ABB RobotStudio station: powerpac.rsstn

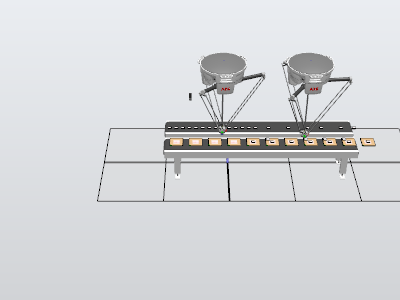
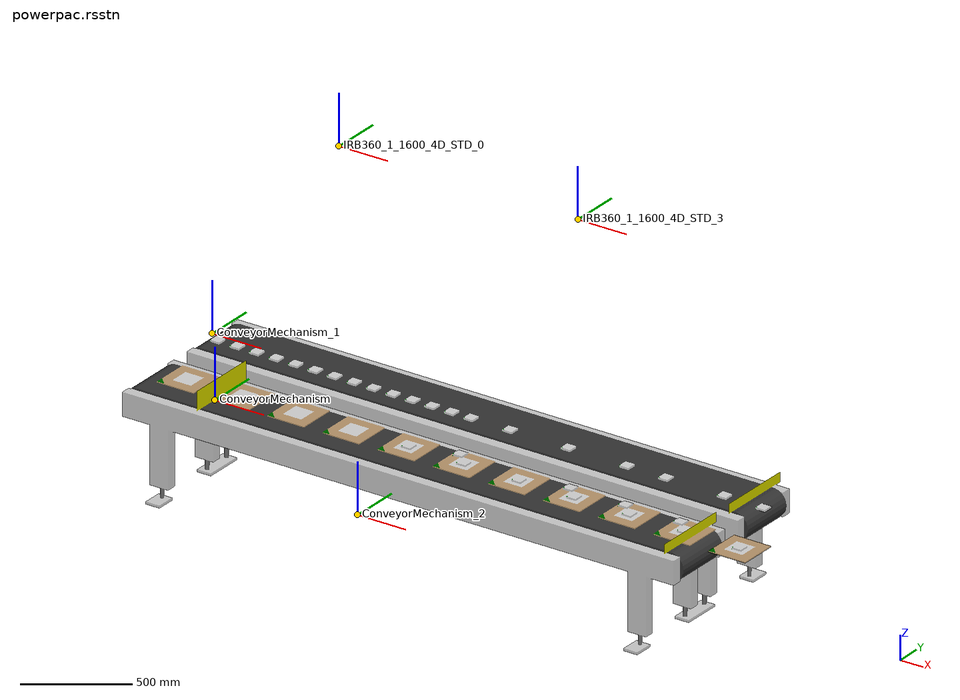
[picture v1: parts stored in the station drawn from their meshes, with robot base, taught points and paths (robot models come from the ABB library and are not in the file)]
Station Station (saved by RobotStudio 22.3.10141.1)
Controller Controller5, task T_ROB1: task frame (RAPID world) sits at (1200, 0, 1800) mm in the station
Controller Controller4, task T_ROB1: task frame (RAPID world) sits at (-100, 0, 1800) mm in the station
Controller Controller4
  mechanical unit ROB_1: IRB360_1_1600_4D_STD_02, 4 joints, base frame (0, 0, 0) mm, rotated rx 180 ry 0 rz 0 deg
  mechanical unit CNV2: ConveyorMechanism, 1 joints, base frame (-500, -250, -1300) mm
  mechanical unit CNV1: ConveyorMechanism_1, 1 joints, base frame (-900, 300, -1300) mm
Controller Controller5
  mechanical unit ROB_1: IRB360_1_1600_4D_STD_3, 4 joints, base frame (0, 0, 0) mm, rotated rx 180 ry 0 rz 0 deg
  mechanical unit CNV2: ConveyorMechanism_2, 1 joints, base frame (0, 0, 0) mm
  mechanical unit CNV1: ConveyorMechanism_3, 1 joints, base frame (0, 0, 0) mm
Layout (positions relative to the parent item):
  - IRB360_1_1600_4D_STD_02 [mechanism, from Robots\IRB360_1_1600_4D_STD_02.rslib] at (-100, 0, 1800) mm, rotated rx 180 ry 0 rz 0 deg; joint values [-0.192, -0.192, -0.192, 0] (rad or m)
  - Line [smart component]
      properties: Enabled=true
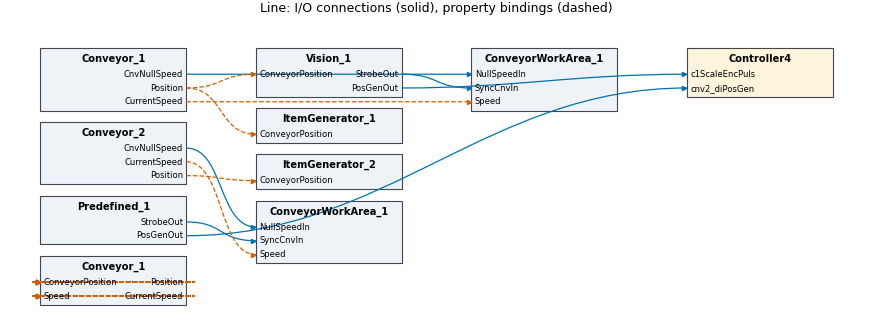
      connections:
        Conveyor_1.CnvNullSpeed -> ConveyorWorkArea_1.NullSpeedIn
        Conveyor_2.CnvNullSpeed -> ConveyorWorkArea_1.NullSpeedIn
        Vision_1.StrobeOut -> ConveyorWorkArea_1.SyncCnvIn
        Vision_1.PosGenOut -> Controller4.c1ScaleEncPuls
        Predefined_1.StrobeOut -> ConveyorWorkArea_1.SyncCnvIn
        Predefined_1.PosGenOut -> Controller4.cnv2_diPosGen
        Conveyor_1.Position => Vision_1.ConveyorPosition
        Conveyor_1.CurrentSpeed => ConveyorWorkArea_1.Speed
        Conveyor_1.Position => ItemGenerator_1.ConveyorPosition
        Conveyor_2.Position => ItemGenerator_2.ConveyorPosition
        Conveyor_1.Position => Vision_1.ConveyorPosition
        Conveyor_1.CurrentSpeed => ConveyorWorkArea_1.Speed
        Conveyor_1.Position => ItemGenerator_1.ConveyorPosition
        Conveyor_2.Position => ItemGenerator_2.ConveyorPosition
        Conveyor_1.Position => Vision_1.ConveyorPosition
        Conveyor_1.CurrentSpeed => ConveyorWorkArea_1.Speed
        Conveyor_2.CurrentSpeed => ConveyorWorkArea_1.Speed
        Conveyor_1.Position => ItemGenerator_1.ConveyorPosition
        Conveyor_2.Position => ItemGenerator_2.ConveyorPosition
        Conveyor_1.Position => Vision_1.ConveyorPosition
        Conveyor_1.CurrentSpeed => ConveyorWorkArea_1.Speed
        Conveyor_2.CurrentSpeed => ConveyorWorkArea_1.Speed
        Conveyor_1.Position => ItemGenerator_1.ConveyorPosition
        Conveyor_2.Position => ItemGenerator_2.ConveyorPosition
        Conveyor_1.Position => Vision_1.ConveyorPosition
        Conveyor_1.CurrentSpeed => ConveyorWorkArea_1.Speed
        Conveyor_2.CurrentSpeed => ConveyorWorkArea_1.Speed
        Conveyor_1.Position => ItemGenerator_1.ConveyorPosition
        Conveyor_2.Position => ItemGenerator_2.ConveyorPosition
        Conveyor_1.Position => Vision_1.ConveyorPosition
        Conveyor_1.CurrentSpeed => ConveyorWorkArea_1.Speed
        Conveyor_2.CurrentSpeed => ConveyorWorkArea_1.Speed
        Conveyor_1.Position => ItemGenerator_1.ConveyorPosition
        Conveyor_2.Position => ItemGenerator_2.ConveyorPosition
    - Job_1 [smart component]
        properties: Project=C:\Users\aedpu\OneDrive\Documents\RobotStudio\Picking\PMPPProject.pmproj; Enabled=true; UserName=admin; Password=password
      - ItemGenerator_1 [smart component]
          properties: ItemSource=Item_1; PositionSource=Vision_1; Conveyor=Conveyor_1; Offset=[[1 0 0 0] [0 1 0 0] [0 0 1 0] [-1 0.250000005960464 0.5 1]]; ObjectLocation=[0.00273041710121014 0 0]; ObjectOrientation=[0 0 0]; ItemContainer=MotionContainer; ConveyorPosition=8.22780232501204; TriggerDistance=0.105999998748302; ProductInfos=1 True 0 0 0 0 0 0;; Repeat=true; Stability=100; OrientationStability=100; ZOriDevMin=0; ZOriDevMax=0; RejectionRatio=0; PositionStability=100; XPosDevMin=0; XPosDevMax=0; YPosDevMin=0; YPosDevMax=0
          signals: DO ItemCreated, DI ItemCopied, DI QueueIdleIn, DI GenerateItemsIn, DO GenerateItemsOut, DI GenerateMultipleItemsIn
          connections:
            ItemGenerator_1.GenerateItemsIn -> ItemGenerator_1.GenerateItemsOut
            ItemGenerator_1.GenerateItemsOut -> ItemCopier.Execute
            ItemCopier.Executed -> ItemGenerator_1.ItemCopied
            ItemCopier.Executed -> ItemCounter.Increase
            CountComparer.Output -> ItemGenerator_1.ItemCreated
            ItemGenerator_1.QueueIdleIn -> Inverter.Input
            Inverter.OutputLow -> ItemCounter.Reset
            ItemGenerator_1.ItemSource => ItemCopier.Source
            ItemGenerator_1.ItemContainer => ItemCopier.Parent
            ItemCounter.Count => CountComparer.ValueA
        - ItemCopier [smart component, from Components\Source.rslib]
            properties: Source=Item_1; Copy=Item_1_1803; Parent=MotionContainer; Position=[0 0 0]; Orientation=[0 0 0]; Transient=false; PhysicsBehavior=0
        - ItemCounter [smart component, from Components\Counter.rslib]
            properties: Count=77
        - CountComparer [smart component, from Components\Comparer.rslib]
            properties: ValueA=77; Operator=>; ValueB=0
        - Inverter [smart component, from Components\LogicSplit.rslib]
      - ItemGenerator_2 [smart component]
          properties: ItemSource=Container_1; PositionSource=Predefined_1; Conveyor=Conveyor_2; Offset=[[1 0 0 0] [0 1 0 0] [0 0 1 0] [-1 -0.249999994039536 0.5 1]]; ObjectLocation=[0.00292999639970226 0 0]; ObjectOrientation=[0 0 0]; ItemContainer=MotionContainer; ConveyorPosition=8.18460232329542; TriggerDistance=0.300000011920929; ProductInfos=1 True 0 0 0 0 0 0;; Repeat=true; Stability=100; OrientationStability=100; ZOriDevMin=0; ZOriDevMax=0; RejectionRatio=0; PositionStability=100; XPosDevMin=0; XPosDevMax=0; YPosDevMin=0; YPosDevMax=0
          signals: DO ItemCreated, DI ItemCopied, DI QueueIdleIn, DI GenerateItemsIn, DO GenerateItemsOut, DI GenerateMultipleItemsIn
          connections:
            ItemGenerator_2.GenerateItemsIn -> ItemGenerator_2.GenerateItemsOut
            ItemGenerator_2.GenerateItemsOut -> ItemCopier.Execute
            ItemCopier.Executed -> ItemGenerator_2.ItemCopied
            ItemCopier.Executed -> ItemCounter.Increase
            CountComparer.Output -> ItemGenerator_2.ItemCreated
            ItemGenerator_2.QueueIdleIn -> Inverter.Input
            Inverter.OutputLow -> ItemCounter.Reset
            ItemGenerator_2.ItemSource => ItemCopier.Source
            ItemGenerator_2.ItemContainer => ItemCopier.Parent
            ItemCounter.Count => CountComparer.ValueA
        - ItemCopier [smart component, from Components\Source.rslib]
            properties: Source=Container_1; Copy=Container_1_1804; Parent=MotionContainer; Position=[0 0 0]; Orientation=[0 0 0]; Transient=false; PhysicsBehavior=0
        - ItemCounter [smart component, from Components\Counter.rslib]
            properties: Count=27
        - CountComparer [smart component, from Components\Comparer.rslib]
            properties: ValueA=27; Operator=>; ValueB=0
        - Inverter [smart component, from Components\LogicSplit.rslib]
    - PickPlaceTool_1 [smart component, from %3FC1A3B3-DC1B-42D2-8AA6-D9E1B3C46536%\PMPickPlaceTool.rslib] at (-100, 0, 623.14) mm, rotated rx 180 ry 0 rz 0 deg
        properties: AttachLocation=[0 0 0.07]; AttachOrientation=[3.14159265358979 0 0]; PickLimit=0.05; PlaceLimit=0.1; GripSignal=doVacuum1; ReleaseSignal=doBlow1
        connections:
          PickPlaceTool_1.GripIn -> PickPlaceTool_1.GripOut
          PickPlaceTool_1.ReleaseIn -> PickPlaceTool_1.ReleaseOut
    - PickPlaceTool_2 [smart component, from %3FC1A3B3-DC1B-42D2-8AA6-D9E1B3C46536%\PMPickPlaceTool.rslib] at (1200, 0, 545.63) mm, rotated rx 180 ry 0 rz 0 deg
        properties: AttachLocation=[0 0 0.07]; AttachOrientation=[3.14159265358979 0 0]; PickLimit=0.05; PlaceLimit=0.1; GripSignal=doVacuum1; ReleaseSignal=doBlow1
        connections:
          PickPlaceTool_2.GripIn -> PickPlaceTool_2.GripOut
          PickPlaceTool_2.ReleaseIn -> PickPlaceTool_2.ReleaseOut
    - Vision_1 [smart component, from %3FC1A3B3-DC1B-42D2-8AA6-D9E1B3C46536%\PMVision.rslib] at (-600, 300, 1000) mm
        properties: Id=213262b1-3477-4070-b768-c16ae12cfddf; Entry=-0.2; Exit=0.2; Left=-0.2; Right=0.2; LimitVisionWidth=false; TriggerType=Distance; TriggerDistance=0.150000005960464; PositionDelay=0; ConveyorPosition=8.22780232501204; SpotLight=Camera 1; PlaneSensor=(none)
        connections:
          Vision_1.TrigVisionIn -> Vision_1.StrobeOut
          Vision_1.PosGenIn -> Vision_1.PosGenOut
    - Conveyor_1 [smart component] at (-1000, 300, 500) mm
        properties: CalibrationLocation=[0 0 0]; CalibrationOrientation=[0 0 0]; Length=3; Width=0.400000005960464; Exit=3; Speed=0.300000011920929; Acc=0.5; Dec=1; CurrentSpeed=0; Position=8.22780232501204; SpeedSignal=; IOMapSystemId=
        signals: DI CnvStartStopIn, DO CnvStartStopOut, DO CnvNullSpeed, AI CnvSpeed
        connections:
          Conveyor_1.CnvStartStopIn -> Conveyor_1.CnvStartStopOut
          ConveyorWorkArea_1.Cnt1FromEncOut -> Controller4.CNV1_giCntSim
          ConveyorWorkArea_1.ConnectedOut -> Controller4.c1Connected
          ConveyorWorkArea_1.NewObjStrobeOut -> Controller4.c1NewObjStrobe
          ConveyorWorkArea_1.PositionOut -> Controller4.c1Position
          ConveyorWorkArea_1.SpeedOut -> Controller4.c1Speed
          ConveyorWorkArea_1.NullSpeedOut -> Controller4.c1NullSpeed
          Conveyor_1.CurrentSpeed => Mover.Speed
          Conveyor_1.Exit => ExitHandler.Transform.X
      - MotionContainer [graphiccomponentgroup] at (8227.8, 0, 0) mm
        - Item_1_1766 [smart component] at (-5194, -50, 0) mm
            properties: Id=2704d276-ea2d-4d5a-9f22-027de52e7f75; GripLocation=[0 0 0.01]; GripOrientation=[0 0 0]; Assembled=true; Detect=true; Accepted=true; IgnoreOrientation=false
          - Item1 [graphiccomponentgroup]
            - MainBody [part], size 50 x 50 x 10 mm
            - OuterLine [part], size 50 x 50 x 10 mm
            - Labels [part], size 25 x 25 x 0 mm
            - Origin [part], size 10.5 x 10.5 x 11 mm
            - RejectSymbol [part], size 23.8 x 48.1 x 1 mm
        - Item_1_1768 [smart component] at (-5406, -50, 0) mm
            properties: Id=2704d276-ea2d-4d5a-9f22-027de52e7f75; GripLocation=[0 0 0.01]; GripOrientation=[0 0 0]; Assembled=true; Detect=true; Accepted=true; IgnoreOrientation=false
          - Item1 [graphiccomponentgroup]
            - MainBody [part], size 50 x 50 x 10 mm
            - OuterLine [part], size 50 x 50 x 10 mm
            - Labels [part], size 25 x 25 x 0 mm
            - Origin [part], size 10.5 x 10.5 x 11 mm
            - RejectSymbol [part], size 23.8 x 48.1 x 1 mm
        - Item_1_1772 [smart component] at (-5724, -50, 0) mm
            properties: Id=2704d276-ea2d-4d5a-9f22-027de52e7f75; GripLocation=[0 0 0.01]; GripOrientation=[0 0 0]; Assembled=true; Detect=true; Accepted=true; IgnoreOrientation=false
          - Item1 [graphiccomponentgroup]
            - MainBody [part], size 50 x 50 x 10 mm
            - OuterLine [part], size 50 x 50 x 10 mm
            - Labels [part], size 25 x 25 x 0 mm
            - Origin [part], size 10.5 x 10.5 x 11 mm
            - RejectSymbol [part], size 23.8 x 48.1 x 1 mm
        - Item_1_1775 [smart component] at (-5936, -50, 0) mm
            properties: Id=2704d276-ea2d-4d5a-9f22-027de52e7f75; GripLocation=[0 0 0.01]; GripOrientation=[0 0 0]; Assembled=true; Detect=true; Accepted=true; IgnoreOrientation=false
          - Item1 [graphiccomponentgroup]
            - MainBody [part], size 50 x 50 x 10 mm
            - OuterLine [part], size 50 x 50 x 10 mm
            - Labels [part], size 25 x 25 x 0 mm
            - Origin [part], size 10.5 x 10.5 x 11 mm
            - RejectSymbol [part], size 23.8 x 48.1 x 1 mm
        - Item_1_1779 [smart component] at (-6254, -50, 0) mm
            properties: Id=2704d276-ea2d-4d5a-9f22-027de52e7f75; GripLocation=[0 0 0.01]; GripOrientation=[0 0 0]; Assembled=true; Detect=true; Accepted=true; IgnoreOrientation=false
          - Item1 [graphiccomponentgroup]
            - MainBody [part], size 50 x 50 x 10 mm
            - OuterLine [part], size 50 x 50 x 10 mm
            - Labels [part], size 25 x 25 x 0 mm
            - Origin [part], size 10.5 x 10.5 x 11 mm
            - RejectSymbol [part], size 23.8 x 48.1 x 1 mm
        - Item_1_1783 [smart component] at (-6572, -50, 0) mm
            properties: Id=2704d276-ea2d-4d5a-9f22-027de52e7f75; GripLocation=[0 0 0.01]; GripOrientation=[0 0 0]; Assembled=true; Detect=true; Accepted=true; IgnoreOrientation=false
          - Item1 [graphiccomponentgroup]
            - MainBody [part], size 50 x 50 x 10 mm
            - OuterLine [part], size 50 x 50 x 10 mm
            - Labels [part], size 25 x 25 x 0 mm
            - Origin [part], size 10.5 x 10.5 x 11 mm
            - RejectSymbol [part], size 23.8 x 48.1 x 1 mm
        - Item_1_1786 [smart component] at (-6784, -50, 0) mm
            properties: Id=2704d276-ea2d-4d5a-9f22-027de52e7f75; GripLocation=[0 0 0.01]; GripOrientation=[0 0 0]; Assembled=true; Detect=true; Accepted=true; IgnoreOrientation=false
          - Item1 [graphiccomponentgroup]
            - MainBody [part], size 50 x 50 x 10 mm
            - OuterLine [part], size 50 x 50 x 10 mm
            - Labels [part], size 25 x 25 x 0 mm
            - Origin [part], size 10.5 x 10.5 x 11 mm
            - RejectSymbol [part], size 23.8 x 48.1 x 1 mm
        - Item_1_1787 [smart component] at (-6890, -50, 0) mm
            properties: Id=2704d276-ea2d-4d5a-9f22-027de52e7f75; GripLocation=[0 0 0.01]; GripOrientation=[0 0 0]; Assembled=true; Detect=true; Accepted=true; IgnoreOrientation=false
          - Item1 [graphiccomponentgroup]
            - MainBody [part], size 50 x 50 x 10 mm
            - OuterLine [part], size 50 x 50 x 10 mm
            - Labels [part], size 25 x 25 x 0 mm
            - Origin [part], size 10.5 x 10.5 x 11 mm
            - RejectSymbol [part], size 23.8 x 48.1 x 1 mm
        - Item_1_1789 [smart component] at (-6996, -50, 0) mm
            properties: Id=2704d276-ea2d-4d5a-9f22-027de52e7f75; GripLocation=[0 0 0.01]; GripOrientation=[0 0 0]; Assembled=true; Detect=true; Accepted=true; IgnoreOrientation=false
          - Item1 [graphiccomponentgroup]
            - MainBody [part], size 50 x 50 x 10 mm
            - OuterLine [part], size 50 x 50 x 10 mm
            - Labels [part], size 25 x 25 x 0 mm
            - Origin [part], size 10.5 x 10.5 x 11 mm
            - RejectSymbol [part], size 23.8 x 48.1 x 1 mm
        - Item_1_1790 [smart component] at (-7102, -50, 0) mm
            properties: Id=2704d276-ea2d-4d5a-9f22-027de52e7f75; GripLocation=[0 0 0.01]; GripOrientation=[0 0 0]; Assembled=true; Detect=true; Accepted=true; IgnoreOrientation=false
          - Item1 [graphiccomponentgroup]
            - MainBody [part], size 50 x 50 x 10 mm
            - OuterLine [part], size 50 x 50 x 10 mm
            - Labels [part], size 25 x 25 x 0 mm
            - Origin [part], size 10.5 x 10.5 x 11 mm
            - RejectSymbol [part], size 23.8 x 48.1 x 1 mm
        - Item_1_1791 [smart component] at (-7208, -50, 0) mm
            properties: Id=2704d276-ea2d-4d5a-9f22-027de52e7f75; GripLocation=[0 0 0.01]; GripOrientation=[0 0 0]; Assembled=true; Detect=true; Accepted=true; IgnoreOrientation=false
          - Item1 [graphiccomponentgroup]
            - MainBody [part], size 50 x 50 x 10 mm
            - OuterLine [part], size 50 x 50 x 10 mm
            - Labels [part], size 25 x 25 x 0 mm
            - Origin [part], size 10.5 x 10.5 x 11 mm
            - RejectSymbol [part], size 23.8 x 48.1 x 1 mm
        - Item_1_1793 [smart component] at (-7314, -50, 0) mm
            properties: Id=2704d276-ea2d-4d5a-9f22-027de52e7f75; GripLocation=[0 0 0.01]; GripOrientation=[0 0 0]; Assembled=true; Detect=true; Accepted=true; IgnoreOrientation=false
          - Item1 [graphiccomponentgroup]
            - MainBody [part], size 50 x 50 x 10 mm
            - OuterLine [part], size 50 x 50 x 10 mm
            - Labels [part], size 25 x 25 x 0 mm
            - Origin [part], size 10.5 x 10.5 x 11 mm
            - RejectSymbol [part], size 23.8 x 48.1 x 1 mm
        - Item_1_1794 [smart component] at (-7420, -50, 0) mm
            properties: Id=2704d276-ea2d-4d5a-9f22-027de52e7f75; GripLocation=[0 0 0.01]; GripOrientation=[0 0 0]; Assembled=true; Detect=true; Accepted=true; IgnoreOrientation=false
          - Item1 [graphiccomponentgroup]
            - MainBody [part], size 50 x 50 x 10 mm
            - OuterLine [part], size 50 x 50 x 10 mm
            - Labels [part], size 25 x 25 x 0 mm
            - Origin [part], size 10.5 x 10.5 x 11 mm
            - RejectSymbol [part], size 23.8 x 48.1 x 1 mm
        - Item_1_1795 [smart component] at (-7526, -50, 0) mm
            properties: Id=2704d276-ea2d-4d5a-9f22-027de52e7f75; GripLocation=[0 0 0.01]; GripOrientation=[0 0 0]; Assembled=true; Detect=true; Accepted=true; IgnoreOrientation=false
          - Item1 [graphiccomponentgroup]
            - MainBody [part], size 50 x 50 x 10 mm
            - OuterLine [part], size 50 x 50 x 10 mm
            - Labels [part], size 25 x 25 x 0 mm
            - Origin [part], size 10.5 x 10.5 x 11 mm
            - RejectSymbol [part], size 23.8 x 48.1 x 1 mm
        - Item_1_1797 [smart component] at (-7632, -50, 0) mm
            properties: Id=2704d276-ea2d-4d5a-9f22-027de52e7f75; GripLocation=[0 0 0.01]; GripOrientation=[0 0 0]; Assembled=true; Detect=true; Accepted=true; IgnoreOrientation=false
          - Item1 [graphiccomponentgroup]
            - MainBody [part], size 50 x 50 x 10 mm
            - OuterLine [part], size 50 x 50 x 10 mm
            - Labels [part], size 25 x 25 x 0 mm
            - Origin [part], size 10.5 x 10.5 x 11 mm
            - RejectSymbol [part], size 23.8 x 48.1 x 1 mm
        - Item_1_1798 [smart component] at (-7738, -50, 0) mm
            properties: Id=2704d276-ea2d-4d5a-9f22-027de52e7f75; GripLocation=[0 0 0.01]; GripOrientation=[0 0 0]; Assembled=true; Detect=true; Accepted=true; IgnoreOrientation=false
          - Item1 [graphiccomponentgroup]
            - MainBody [part], size 50 x 50 x 10 mm
            - OuterLine [part], size 50 x 50 x 10 mm
            - Labels [part], size 25 x 25 x 0 mm
            - Origin [part], size 10.5 x 10.5 x 11 mm
            - RejectSymbol [part], size 23.8 x 48.1 x 1 mm
        - Item_1_1799 [smart component] at (-7844, -50, 0) mm
            properties: Id=2704d276-ea2d-4d5a-9f22-027de52e7f75; GripLocation=[0 0 0.01]; GripOrientation=[0 0 0]; Assembled=true; Detect=true; Accepted=true; IgnoreOrientation=false
          - Item1 [graphiccomponentgroup]
            - MainBody [part], size 50 x 50 x 10 mm
            - OuterLine [part], size 50 x 50 x 10 mm
            - Labels [part], size 25 x 25 x 0 mm
            - Origin [part], size 10.5 x 10.5 x 11 mm
            - RejectSymbol [part], size 23.8 x 48.1 x 1 mm
        - Item_1_1801 [smart component] at (-7950, -50, 0) mm
            properties: Id=2704d276-ea2d-4d5a-9f22-027de52e7f75; GripLocation=[0 0 0.01]; GripOrientation=[0 0 0]; Assembled=true; Detect=true; Accepted=true; IgnoreOrientation=false
          - Item1 [graphiccomponentgroup]
            - MainBody [part], size 50 x 50 x 10 mm
            - OuterLine [part], size 50 x 50 x 10 mm
            - Labels [part], size 25 x 25 x 0 mm
            - Origin [part], size 10.5 x 10.5 x 11 mm
            - RejectSymbol [part], size 23.8 x 48.1 x 1 mm
        - Item_1_1802 [smart component] at (-8056, -50, 0) mm
            properties: Id=2704d276-ea2d-4d5a-9f22-027de52e7f75; GripLocation=[0 0 0.01]; GripOrientation=[0 0 0]; Assembled=true; Detect=true; Accepted=true; IgnoreOrientation=false
          - Item1 [graphiccomponentgroup]
            - MainBody [part], size 50 x 50 x 10 mm
            - OuterLine [part], size 50 x 50 x 10 mm
            - Labels [part], size 25 x 25 x 0 mm
            - Origin [part], size 10.5 x 10.5 x 11 mm
            - RejectSymbol [part], size 23.8 x 48.1 x 1 mm
        - Item_1_1803 [smart component] at (-8162, -50, 0) mm
            properties: Id=2704d276-ea2d-4d5a-9f22-027de52e7f75; GripLocation=[0 0 0.01]; GripOrientation=[0 0 0]; Assembled=true; Detect=true; Accepted=true; IgnoreOrientation=false
          - Item1 [graphiccomponentgroup]
            - MainBody [part], size 50 x 50 x 10 mm
            - OuterLine [part], size 50 x 50 x 10 mm
            - Labels [part], size 25 x 25 x 0 mm
            - Origin [part], size 10.5 x 10.5 x 11 mm
            - RejectSymbol [part], size 23.8 x 48.1 x 1 mm
      - Mover [smart component, from Components\LinearMover.rslib]
          properties: Object=MotionContainer; Direction=[0.001 0 0]; Speed=0; Reference=Local; ReferenceObject=(none)
      - ExitHandler [smart component, from %3FC1A3B3-DC1B-42D2-8AA6-D9E1B3C46536%\PMExitHandler.rslib] at (3000, 0, 0) mm
          properties: Count=32; SensedObject=(none)
          connections:
            Timer.Output -> ExitHandler.Execute
        - Timer [smart component, from Components\Timer.rslib]
            properties: StartTime=0; Interval=1; Repeat=true; CurrentTime=32.64
      - ConveyorWorkArea_1 [smart component, from %3FC1A3B3-DC1B-42D2-8AA6-D9E1B3C46536%\PMConveyorWorkArea.rslib]
          properties: WorkAreaType=Pick; PositionSource=Vision_1; PositionGeneratorSignal=cnv1_diPosGen; TrigVisionSignal=cnv1_doTrigVis; CnvStartStopSignal=cnv1_doStartCnv; ControllerMechUnit=CNV1; SystemId={3445A632-8DB2-4EAE-9C35-B4E87A875A90}; Speed=0; QueueIdleSignal=cnv1_doQIdle; CountsPerMeter=20000
          connections:
            Converter.AnalogOutput -> ConveyorWorkArea_1.SpeedIn
            ConveyorWorkArea_1.SpeedIn -> ConveyorWorkArea_1.SpeedOut
            ConveyorWorkArea_1.NullSpeedIn -> ConveyorWorkArea_1.NullSpeedOut
            ConveyorWorkArea_1.Speed => Converter.AnalogProperty
        - Converter [smart component, from Components\Converter.rslib]
            properties: AnalogProperty=0; DigitalProperty=0; BooleanProperty=false; GroupProperty=0
    - Predefined_1 [smart component, from %3FC1A3B3-DC1B-42D2-8AA6-D9E1B3C46536%\PMPredefined.rslib]
        properties: Id=fbd0e5b6-92fc-4816-a2a1-f9a7d29e2a65; TriggerType=IO; TriggerDistance=0; ConveyorPosition=0; PlaneSensor=PlaneSensor
        connections:
          Predefined_1.PosGenIn -> Predefined_1.PosGenOut
          Predefined_1.PosGenIn -> Predefined_1.StrobeOut
    - Conveyor_2 [smart component] at (-1000, -200, 500) mm
        properties: CalibrationLocation=[0 0 0]; CalibrationOrientation=[0 0 0]; Length=3; Width=0.400000005960464; Exit=3; Speed=0.300000011920929; Acc=0.5; Dec=1; CurrentSpeed=0; Position=8.18460232329542; SpeedSignal=; IOMapSystemId=
        signals: DI CnvStartStopIn, DO CnvStartStopOut, DO CnvNullSpeed, AI CnvSpeed
        connections:
          Conveyor_2.CnvStartStopIn -> Conveyor_2.CnvStartStopOut
          ConveyorWorkArea_1.Cnt1FromEncOut -> Controller4.CNV2_giCntSim
          ConveyorWorkArea_1.ConnectedOut -> Controller4.c2Connected
          ConveyorWorkArea_1.NewObjStrobeOut -> Controller4.c2NewObjStrobe
          ConveyorWorkArea_1.PositionOut -> Controller4.c2Position
          ConveyorWorkArea_1.SpeedOut -> Controller4.c2Speed
          ConveyorWorkArea_1.NullSpeedOut -> Controller4.c2NullSpeed
          Conveyor_2.CurrentSpeed => Mover.Speed
          Conveyor_2.Exit => ExitHandler.Transform.X
      - MotionContainer [graphiccomponentgroup] at (8184.6, 0, 0) mm
        - Container_1_1765 [smart component] at (-5100, -50, 0) mm
            properties: Id=73001933-2678-449b-9029-7b770ab6b154; GripLocation=[0.1 0.1 0.1]; GripOrientation=[0 0 0]; Detect=true; Accepted=true; IgnoreOrientation=false
          - Container1 [graphiccomponentgroup]
            - MainBody [part], size 200 x 200 x 5 mm
            - OuterLine [part], size 200 x 200 x 5 mm
            - Labels [part], size 100 x 100 x 0 mm
            - Origin [part], size 40.5 x 40.5 x 6 mm
            - RejectSymbol [part], size 47.5 x 96.2 x 1 mm
          - Layer_1 [smart component, from %3FC1A3B3-DC1B-42D2-8AA6-D9E1B3C46536%\PMLayer.rslib] at (0, 0, 5) mm
              properties: Pattern=Pattern_1
          - Layer_2 [smart component, from %3FC1A3B3-DC1B-42D2-8AA6-D9E1B3C46536%\PMLayer.rslib] at (0, 0, 15) mm
              properties: Pattern=Pattern_2
          - Item_1_1763 [smart component] at (101.26, 97.68, 5) mm
              properties: Id=2704d276-ea2d-4d5a-9f22-027de52e7f75; GripLocation=[0 0 0.01]; GripOrientation=[0 0 0]; Assembled=true; Detect=true; Accepted=true; IgnoreOrientation=false
            - Item1 [graphiccomponentgroup]
              - MainBody [part], size 50 x 50 x 10 mm
              - OuterLine [part], size 50 x 50 x 10 mm
              - Labels [part], size 25 x 25 x 0 mm
              - Origin [part], size 10.5 x 10.5 x 11 mm
              - RejectSymbol [part], size 23.8 x 48.1 x 1 mm
        - Container_1_1769 [smart component] at (-5400, -50, 0) mm
            properties: Id=73001933-2678-449b-9029-7b770ab6b154; GripLocation=[0.1 0.1 0.1]; GripOrientation=[0 0 0]; Detect=true; Accepted=true; IgnoreOrientation=false
          - Container1 [graphiccomponentgroup]
            - MainBody [part], size 200 x 200 x 5 mm
            - OuterLine [part], size 200 x 200 x 5 mm
            - Labels [part], size 100 x 100 x 0 mm
            - Origin [part], size 40.5 x 40.5 x 6 mm
            - RejectSymbol [part], size 47.5 x 96.2 x 1 mm
          - Layer_1 [smart component, from %3FC1A3B3-DC1B-42D2-8AA6-D9E1B3C46536%\PMLayer.rslib] at (0, 0, 5) mm
              properties: Pattern=Pattern_1
          - Layer_2 [smart component, from %3FC1A3B3-DC1B-42D2-8AA6-D9E1B3C46536%\PMLayer.rslib] at (0, 0, 15) mm
              properties: Pattern=Pattern_2
          - Item_1_1764 [smart component] at (101.26, 97.68, 5) mm
              properties: Id=2704d276-ea2d-4d5a-9f22-027de52e7f75; GripLocation=[0 0 0.01]; GripOrientation=[0 0 0]; Assembled=true; Detect=true; Accepted=true; IgnoreOrientation=false
            - Item1 [graphiccomponentgroup]
              - MainBody [part], size 50 x 50 x 10 mm
              - OuterLine [part], size 50 x 50 x 10 mm
              - Labels [part], size 25 x 25 x 0 mm
              - Origin [part], size 10.5 x 10.5 x 11 mm
              - RejectSymbol [part], size 23.8 x 48.1 x 1 mm
          - Item_1_1767 [smart component] at (35.78, 163, 5) mm
              properties: Id=2704d276-ea2d-4d5a-9f22-027de52e7f75; GripLocation=[0 0 0.01]; GripOrientation=[0 0 0]; Assembled=true; Detect=true; Accepted=true; IgnoreOrientation=false
            - Item1 [graphiccomponentgroup]
              - MainBody [part], size 50 x 50 x 10 mm
              - OuterLine [part], size 50 x 50 x 10 mm
              - Labels [part], size 25 x 25 x 0 mm
              - Origin [part], size 10.5 x 10.5 x 11 mm
              - RejectSymbol [part], size 23.8 x 48.1 x 1 mm
        - Container_1_1773 [smart component] at (-5700, -50, 0) mm
            properties: Id=73001933-2678-449b-9029-7b770ab6b154; GripLocation=[0.1 0.1 0.1]; GripOrientation=[0 0 0]; Detect=true; Accepted=true; IgnoreOrientation=false
          - Container1 [graphiccomponentgroup]
            - MainBody [part], size 200 x 200 x 5 mm
            - OuterLine [part], size 200 x 200 x 5 mm
            - Labels [part], size 100 x 100 x 0 mm
            - Origin [part], size 40.5 x 40.5 x 6 mm
            - RejectSymbol [part], size 47.5 x 96.2 x 1 mm
          - Layer_1 [smart component, from %3FC1A3B3-DC1B-42D2-8AA6-D9E1B3C46536%\PMLayer.rslib] at (0, 0, 5) mm
              properties: Pattern=Pattern_1
          - Layer_2 [smart component, from %3FC1A3B3-DC1B-42D2-8AA6-D9E1B3C46536%\PMLayer.rslib] at (0, 0, 15) mm
              properties: Pattern=Pattern_2
          - Item_1_1770 [smart component] at (101.26, 97.68, 5) mm
              properties: Id=2704d276-ea2d-4d5a-9f22-027de52e7f75; GripLocation=[0 0 0.01]; GripOrientation=[0 0 0]; Assembled=true; Detect=true; Accepted=true; IgnoreOrientation=false
            - Item1 [graphiccomponentgroup]
              - MainBody [part], size 50 x 50 x 10 mm
              - OuterLine [part], size 50 x 50 x 10 mm
              - Labels [part], size 25 x 25 x 0 mm
              - Origin [part], size 10.5 x 10.5 x 11 mm
              - RejectSymbol [part], size 23.8 x 48.1 x 1 mm
          - Item_1_1771 [smart component] at (35.78, 163, 5) mm
              properties: Id=2704d276-ea2d-4d5a-9f22-027de52e7f75; GripLocation=[0 0 0.01]; GripOrientation=[0 0 0]; Assembled=true; Detect=true; Accepted=true; IgnoreOrientation=false
            - Item1 [graphiccomponentgroup]
              - MainBody [part], size 50 x 50 x 10 mm
              - OuterLine [part], size 50 x 50 x 10 mm
              - Labels [part], size 25 x 25 x 0 mm
              - Origin [part], size 10.5 x 10.5 x 11 mm
              - RejectSymbol [part], size 23.8 x 48.1 x 1 mm
        - Container_1_1777 [smart component] at (-6000, -50, 0) mm
            properties: Id=73001933-2678-449b-9029-7b770ab6b154; GripLocation=[0.1 0.1 0.1]; GripOrientation=[0 0 0]; Detect=true; Accepted=true; IgnoreOrientation=false
          - Container1 [graphiccomponentgroup]
            - MainBody [part], size 200 x 200 x 5 mm
            - OuterLine [part], size 200 x 200 x 5 mm
            - Labels [part], size 100 x 100 x 0 mm
            - Origin [part], size 40.5 x 40.5 x 6 mm
            - RejectSymbol [part], size 47.5 x 96.2 x 1 mm
          - Layer_1 [smart component, from %3FC1A3B3-DC1B-42D2-8AA6-D9E1B3C46536%\PMLayer.rslib] at (0, 0, 5) mm
              properties: Pattern=Pattern_1
          - Layer_2 [smart component, from %3FC1A3B3-DC1B-42D2-8AA6-D9E1B3C46536%\PMLayer.rslib] at (0, 0, 15) mm
              properties: Pattern=Pattern_2
          - Item_1_1774 [smart component] at (101.26, 97.68, 5) mm
              properties: Id=2704d276-ea2d-4d5a-9f22-027de52e7f75; GripLocation=[0 0 0.01]; GripOrientation=[0 0 0]; Assembled=true; Detect=true; Accepted=true; IgnoreOrientation=false
            - Item1 [graphiccomponentgroup]
              - MainBody [part], size 50 x 50 x 10 mm
              - OuterLine [part], size 50 x 50 x 10 mm
              - Labels [part], size 25 x 25 x 0 mm
              - Origin [part], size 10.5 x 10.5 x 11 mm
              - RejectSymbol [part], size 23.8 x 48.1 x 1 mm
          - Item_1_1776 [smart component] at (35.78, 163, 5) mm
              properties: Id=2704d276-ea2d-4d5a-9f22-027de52e7f75; GripLocation=[0 0 0.01]; GripOrientation=[0 0 0]; Assembled=true; Detect=true; Accepted=true; IgnoreOrientation=false
            - Item1 [graphiccomponentgroup]
              - MainBody [part], size 50 x 50 x 10 mm
              - OuterLine [part], size 50 x 50 x 10 mm
              - Labels [part], size 25 x 25 x 0 mm
              - Origin [part], size 10.5 x 10.5 x 11 mm
              - RejectSymbol [part], size 23.8 x 48.1 x 1 mm
        - Container_1_1781 [smart component] at (-6300, -50, 0) mm
            properties: Id=73001933-2678-449b-9029-7b770ab6b154; GripLocation=[0.1 0.1 0.1]; GripOrientation=[0 0 0]; Detect=true; Accepted=true; IgnoreOrientation=false
          - Container1 [graphiccomponentgroup]
            - MainBody [part], size 200 x 200 x 5 mm
            - OuterLine [part], size 200 x 200 x 5 mm
            - Labels [part], size 100 x 100 x 0 mm
            - Origin [part], size 40.5 x 40.5 x 6 mm
            - RejectSymbol [part], size 47.5 x 96.2 x 1 mm
          - Layer_1 [smart component, from %3FC1A3B3-DC1B-42D2-8AA6-D9E1B3C46536%\PMLayer.rslib] at (0, 0, 5) mm
              properties: Pattern=Pattern_1
          - Layer_2 [smart component, from %3FC1A3B3-DC1B-42D2-8AA6-D9E1B3C46536%\PMLayer.rslib] at (0, 0, 15) mm
              properties: Pattern=Pattern_2
          - Item_1_1778 [smart component] at (101.26, 97.68, 5) mm
              properties: Id=2704d276-ea2d-4d5a-9f22-027de52e7f75; GripLocation=[0 0 0.01]; GripOrientation=[0 0 0]; Assembled=true; Detect=true; Accepted=true; IgnoreOrientation=false
            - Item1 [graphiccomponentgroup]
              - MainBody [part], size 50 x 50 x 10 mm
              - OuterLine [part], size 50 x 50 x 10 mm
              - Labels [part], size 25 x 25 x 0 mm
              - Origin [part], size 10.5 x 10.5 x 11 mm
              - RejectSymbol [part], size 23.8 x 48.1 x 1 mm
        - Container_1_1784 [smart component] at (-6600, -50, 0) mm
            properties: Id=73001933-2678-449b-9029-7b770ab6b154; GripLocation=[0.1 0.1 0.1]; GripOrientation=[0 0 0]; Detect=true; Accepted=true; IgnoreOrientation=false
          - Container1 [graphiccomponentgroup]
            - MainBody [part], size 200 x 200 x 5 mm
            - OuterLine [part], size 200 x 200 x 5 mm
            - Labels [part], size 100 x 100 x 0 mm
            - Origin [part], size 40.5 x 40.5 x 6 mm
            - RejectSymbol [part], size 47.5 x 96.2 x 1 mm
          - Layer_1 [smart component, from %3FC1A3B3-DC1B-42D2-8AA6-D9E1B3C46536%\PMLayer.rslib] at (0, 0, 5) mm
              properties: Pattern=Pattern_1
          - Layer_2 [smart component, from %3FC1A3B3-DC1B-42D2-8AA6-D9E1B3C46536%\PMLayer.rslib] at (0, 0, 15) mm
              properties: Pattern=Pattern_2
          - Item_1_1780 [smart component] at (101.26, 97.68, 5) mm
              properties: Id=2704d276-ea2d-4d5a-9f22-027de52e7f75; GripLocation=[0 0 0.01]; GripOrientation=[0 0 0]; Assembled=true; Detect=true; Accepted=true; IgnoreOrientation=false
            - Item1 [graphiccomponentgroup]
              - MainBody [part], size 50 x 50 x 10 mm
              - OuterLine [part], size 50 x 50 x 10 mm
              - Labels [part], size 25 x 25 x 0 mm
              - Origin [part], size 10.5 x 10.5 x 11 mm
              - RejectSymbol [part], size 23.8 x 48.1 x 1 mm
          - Item_1_1782 [smart component] at (35.78, 163, 5) mm
              properties: Id=2704d276-ea2d-4d5a-9f22-027de52e7f75; GripLocation=[0 0 0.01]; GripOrientation=[0 0 0]; Assembled=true; Detect=true; Accepted=true; IgnoreOrientation=false
            - Item1 [graphiccomponentgroup]
              - MainBody [part], size 50 x 50 x 10 mm
              - OuterLine [part], size 50 x 50 x 10 mm
              - Labels [part], size 25 x 25 x 0 mm
              - Origin [part], size 10.5 x 10.5 x 11 mm
              - RejectSymbol [part], size 23.8 x 48.1 x 1 mm
        - Container_1_1788 [smart component] at (-6900, -50, 0) mm
            properties: Id=73001933-2678-449b-9029-7b770ab6b154; GripLocation=[0.1 0.1 0.1]; GripOrientation=[0 0 0]; Detect=true; Accepted=true; IgnoreOrientation=false
          - Container1 [graphiccomponentgroup]
            - MainBody [part], size 200 x 200 x 5 mm
            - OuterLine [part], size 200 x 200 x 5 mm
            - Labels [part], size 100 x 100 x 0 mm
            - Origin [part], size 40.5 x 40.5 x 6 mm
            - RejectSymbol [part], size 47.5 x 96.2 x 1 mm
          - Layer_1 [smart component, from %3FC1A3B3-DC1B-42D2-8AA6-D9E1B3C46536%\PMLayer.rslib] at (0, 0, 5) mm
              properties: Pattern=Pattern_1
          - Layer_2 [smart component, from %3FC1A3B3-DC1B-42D2-8AA6-D9E1B3C46536%\PMLayer.rslib] at (0, 0, 15) mm
              properties: Pattern=Pattern_2
          - Item_1_1785 [smart component] at (101.26, 97.68, 5) mm
              properties: Id=2704d276-ea2d-4d5a-9f22-027de52e7f75; GripLocation=[0 0 0.01]; GripOrientation=[0 0 0]; Assembled=true; Detect=true; Accepted=true; IgnoreOrientation=false
            - Item1 [graphiccomponentgroup]
              - MainBody [part], size 50 x 50 x 10 mm
              - OuterLine [part], size 50 x 50 x 10 mm
              - Labels [part], size 25 x 25 x 0 mm
              - Origin [part], size 10.5 x 10.5 x 11 mm
              - RejectSymbol [part], size 23.8 x 48.1 x 1 mm
        - Container_1_1792 [smart component] at (-7200, -50, 0) mm
            properties: Id=73001933-2678-449b-9029-7b770ab6b154; GripLocation=[0.1 0.1 0.1]; GripOrientation=[0 0 0]; Detect=true; Accepted=true; IgnoreOrientation=false
          - Container1 [graphiccomponentgroup]
            - MainBody [part], size 200 x 200 x 5 mm
            - OuterLine [part], size 200 x 200 x 5 mm
            - Labels [part], size 100 x 100 x 0 mm
            - Origin [part], size 40.5 x 40.5 x 6 mm
            - RejectSymbol [part], size 47.5 x 96.2 x 1 mm
          - Layer_1 [smart component, from %3FC1A3B3-DC1B-42D2-8AA6-D9E1B3C46536%\PMLayer.rslib] at (0, 0, 5) mm
              properties: Pattern=Pattern_1
          - Layer_2 [smart component, from %3FC1A3B3-DC1B-42D2-8AA6-D9E1B3C46536%\PMLayer.rslib] at (0, 0, 15) mm
              properties: Pattern=Pattern_2
        - Container_1_1796 [smart component] at (-7500, -50, 0) mm
            properties: Id=73001933-2678-449b-9029-7b770ab6b154; GripLocation=[0.1 0.1 0.1]; GripOrientation=[0 0 0]; Detect=true; Accepted=true; IgnoreOrientation=false
          - Container1 [graphiccomponentgroup]
            - MainBody [part], size 200 x 200 x 5 mm
            - OuterLine [part], size 200 x 200 x 5 mm
            - Labels [part], size 100 x 100 x 0 mm
            - Origin [part], size 40.5 x 40.5 x 6 mm
            - RejectSymbol [part], size 47.5 x 96.2 x 1 mm
          - Layer_1 [smart component, from %3FC1A3B3-DC1B-42D2-8AA6-D9E1B3C46536%\PMLayer.rslib] at (0, 0, 5) mm
              properties: Pattern=Pattern_1
          - Layer_2 [smart component, from %3FC1A3B3-DC1B-42D2-8AA6-D9E1B3C46536%\PMLayer.rslib] at (0, 0, 15) mm
              properties: Pattern=Pattern_2
        - Container_1_1800 [smart component] at (-7800, -50, 0) mm
            properties: Id=73001933-2678-449b-9029-7b770ab6b154; GripLocation=[0.1 0.1 0.1]; GripOrientation=[0 0 0]; Detect=true; Accepted=true; IgnoreOrientation=false
          - Container1 [graphiccomponentgroup]
            - MainBody [part], size 200 x 200 x 5 mm
            - OuterLine [part], size 200 x 200 x 5 mm
            - Labels [part], size 100 x 100 x 0 mm
            - Origin [part], size 40.5 x 40.5 x 6 mm
            - RejectSymbol [part], size 47.5 x 96.2 x 1 mm
          - Layer_1 [smart component, from %3FC1A3B3-DC1B-42D2-8AA6-D9E1B3C46536%\PMLayer.rslib] at (0, 0, 5) mm
              properties: Pattern=Pattern_1
          - Layer_2 [smart component, from %3FC1A3B3-DC1B-42D2-8AA6-D9E1B3C46536%\PMLayer.rslib] at (0, 0, 15) mm
              properties: Pattern=Pattern_2
        - Container_1_1804 [smart component] at (-8100, -50, 0) mm
            properties: Id=73001933-2678-449b-9029-7b770ab6b154; GripLocation=[0.1 0.1 0.1]; GripOrientation=[0 0 0]; Detect=true; Accepted=true; IgnoreOrientation=false
          - Container1 [graphiccomponentgroup]
            - MainBody [part], size 200 x 200 x 5 mm
            - OuterLine [part], size 200 x 200 x 5 mm
            - Labels [part], size 100 x 100 x 0 mm
            - Origin [part], size 40.5 x 40.5 x 6 mm
            - RejectSymbol [part], size 47.5 x 96.2 x 1 mm
          - Layer_1 [smart component, from %3FC1A3B3-DC1B-42D2-8AA6-D9E1B3C46536%\PMLayer.rslib] at (0, 0, 5) mm
              properties: Pattern=Pattern_1
          - Layer_2 [smart component, from %3FC1A3B3-DC1B-42D2-8AA6-D9E1B3C46536%\PMLayer.rslib] at (0, 0, 15) mm
              properties: Pattern=Pattern_2
      - Mover [smart component, from Components\LinearMover.rslib]
          properties: Object=MotionContainer; Direction=[0.001 0 0]; Speed=0; Reference=Local; ReferenceObject=(none)
      - ExitHandler [smart component, from %3FC1A3B3-DC1B-42D2-8AA6-D9E1B3C46536%\PMExitHandler.rslib] at (3000, 0, 0) mm
          properties: Count=32; SensedObject=(none)
          connections:
            Timer.Output -> ExitHandler.Execute
        - Timer [smart component, from Components\Timer.rslib]
            properties: StartTime=0; Interval=1; Repeat=true; CurrentTime=32.64
      - ConveyorWorkArea_1 [smart component, from %3FC1A3B3-DC1B-42D2-8AA6-D9E1B3C46536%\PMConveyorWorkArea.rslib]
          properties: WorkAreaType=Place; PositionSource=Predefined_1; PositionGeneratorSignal=cnv2_diPosGen; TrigVisionSignal=cnv2_doTrigVis; CnvStartStopSignal=cnv2_doStartCnv; ControllerMechUnit=CNV2; SystemId={3445A632-8DB2-4EAE-9C35-B4E87A875A90}; Speed=0; QueueIdleSignal=cnv2_doQIdle; CountsPerMeter=20000
          connections:
            Converter.AnalogOutput -> ConveyorWorkArea_1.SpeedIn
            ConveyorWorkArea_1.SpeedIn -> ConveyorWorkArea_1.SpeedOut
            ConveyorWorkArea_1.NullSpeedIn -> ConveyorWorkArea_1.NullSpeedOut
            ConveyorWorkArea_1.Speed => Converter.AnalogProperty
        - Converter [smart component, from Components\Converter.rslib]
            properties: AnalogProperty=0; DigitalProperty=0; BooleanProperty=false; GroupProperty=0
    - Item_1 [smart component] at (0, 0, -2011.5) mm
        properties: Id=2704d276-ea2d-4d5a-9f22-027de52e7f75; GripLocation=[0 0 0.01]; GripOrientation=[0 0 0]; Assembled=true; Detect=true; Accepted=true; IgnoreOrientation=false
      - Item1 [graphiccomponentgroup]
        - MainBody [part], size 50 x 50 x 10 mm
        - OuterLine [part], size 50 x 50 x 10 mm
        - Labels [part], size 25 x 25 x 0 mm
        - Origin [part], size 10.5 x 10.5 x 11 mm
        - RejectSymbol [part], size 23.8 x 48.1 x 1 mm
    - Container_1 [smart component] at (0, 0, -2006.5) mm
        properties: Id=73001933-2678-449b-9029-7b770ab6b154; GripLocation=[0.1 0.1 0.1]; GripOrientation=[0 0 0]; Detect=true; Accepted=true; IgnoreOrientation=false
      - Container1 [graphiccomponentgroup]
        - MainBody [part], size 200 x 200 x 5 mm
        - OuterLine [part], size 200 x 200 x 5 mm
        - Labels [part], size 100 x 100 x 0 mm
        - Origin [part], size 40.5 x 40.5 x 6 mm
        - RejectSymbol [part], size 47.5 x 96.2 x 1 mm
      - Layer_1 [smart component, from %3FC1A3B3-DC1B-42D2-8AA6-D9E1B3C46536%\PMLayer.rslib] at (0, 0, 5) mm
          properties: Pattern=Pattern_1
      - Layer_2 [smart component, from %3FC1A3B3-DC1B-42D2-8AA6-D9E1B3C46536%\PMLayer.rslib] at (0, 0, 15) mm
          properties: Pattern=Pattern_2
    - Pattern_1 [smart component, from %3FC1A3B3-DC1B-42D2-8AA6-D9E1B3C46536%\PMPattern.rslib]
        properties: Id=; Positions=0.101258599758148 0.0976838782429695 0 0 0 0 0;0.0357848858460784 0.163001278042793 0 0 0 0 0;0.0357848513871431 0.0375946812331676 0 0 0 0 0;0.161787265539169 0.0393819889053702 0 0 0 0 0;0.161191517114639 0.162405499815941 0 0 0 0 0;
    - Pattern_2 [smart component, from %3FC1A3B3-DC1B-42D2-8AA6-D9E1B3C46536%\PMPattern.rslib]
        properties: Id=; Positions=0.101258599758148 0.0976838782429695 0 0 0 0 0;0.0357848858460784 0.163001278042793 0 0 0 0 0;0.0357848513871431 0.0375946812331676 0 0 0 0 0;0.161787265539169 0.0393819889053702 0 0 0 0 0;0.161191517114639 0.162405499815941 0 0 0 0 0;
  - ConveyorMechanism [mechanism, from %3FC1A3B3-DC1B-42D2-8AA6-D9E1B3C46536%\PMConveyorMechanism.rslib] at (-600, -250, 500) mm
  - ConveyorMechanism_1 [mechanism, from %3FC1A3B3-DC1B-42D2-8AA6-D9E1B3C46536%\PMConveyorMechanism.rslib] at (-1000, 300, 500) mm
  - Vacuum 1x1 [part, from %C4396042-08E9-4F2C-9889-A5FB4C9DA8F9%\Vacuum 1x1.rslib] at (-100, 0, 623.14) mm, rotated rx 180 ry 0 rz 0 deg
  - SC_BeltConveyor [smart component, from %9EFD5320-513E-49BD-B6BC-92403559CEC9%\SC_BeltConveyor.rslib] at (-1000, 100, 0) mm
      properties: ConveyorSpeed=500; FirstLegXpos=0.2; Height=500; LegNumber=1; Length=3000; RollerNumber=31; SourceObject=(none); Width=400
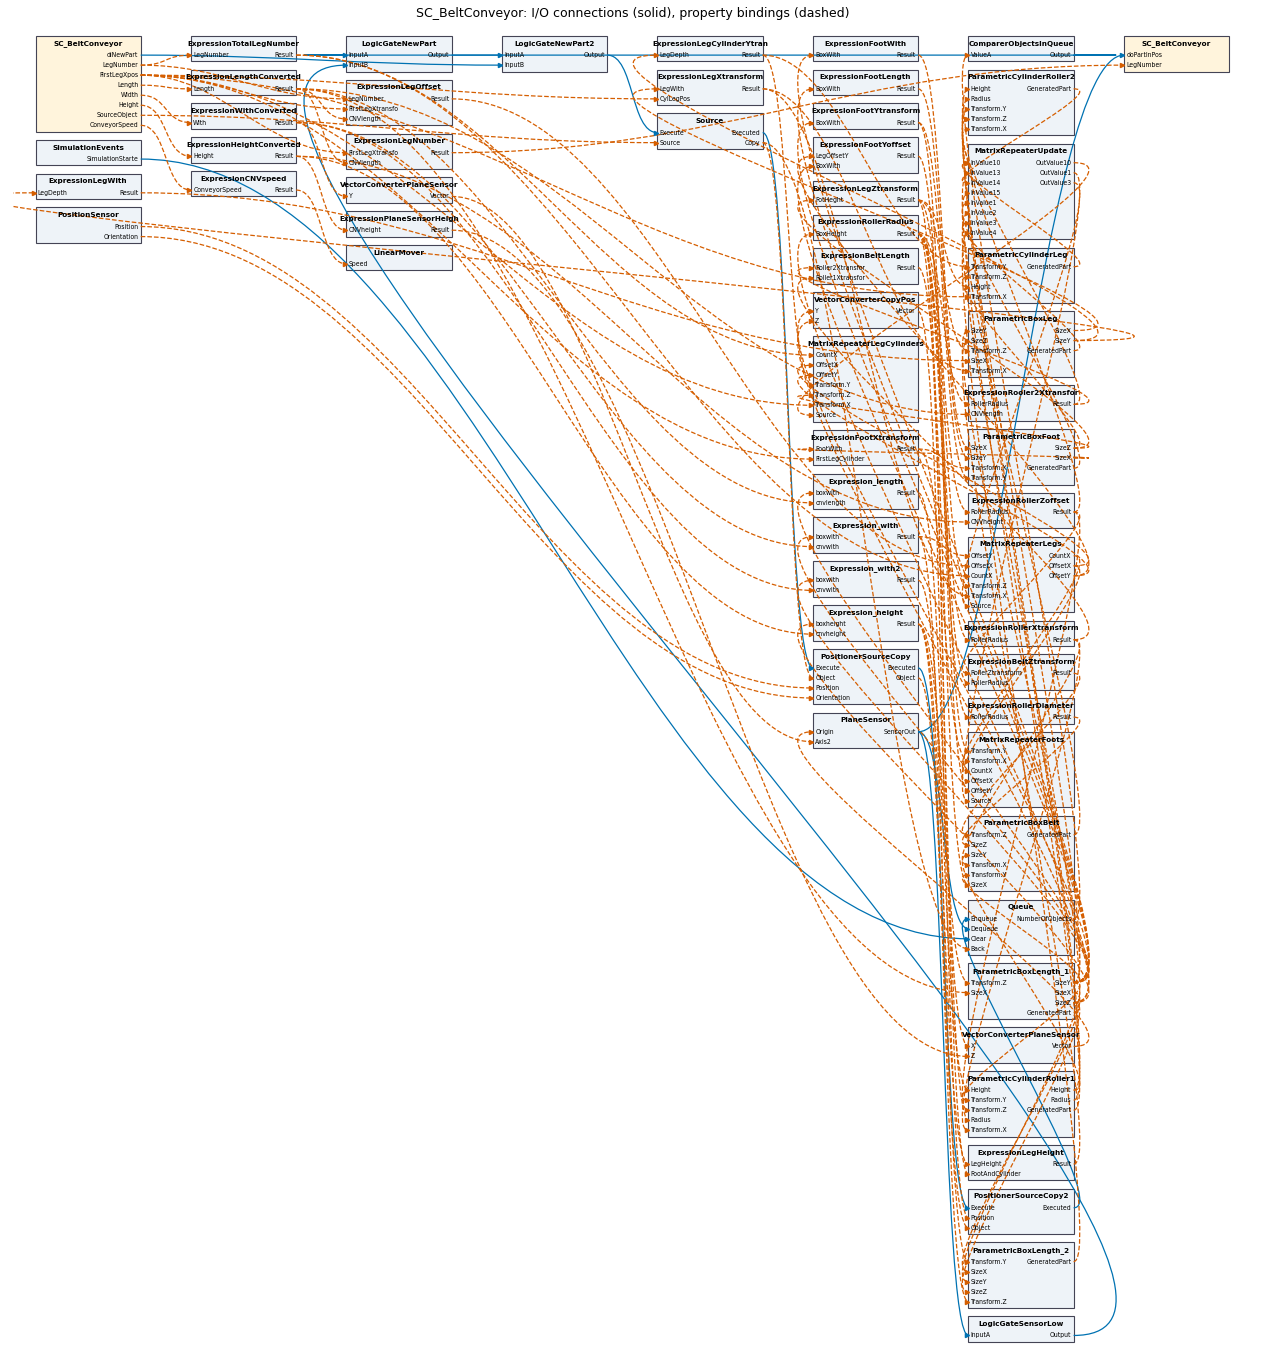
      connections:
        PlaneSensor.SensorOut -> LogicGateSensorLow.InputA
        ComparerObjectsInQueue.Output -> LogicGateNewPart.InputA
        LogicGateSensorLow.Output -> LogicGateNewPart.InputB
        LogicGateNewPart.Output -> LogicGateNewPart2.InputA
        SC_BeltConveyor.diNewPart -> LogicGateNewPart2.InputB
        LogicGateNewPart2.Output -> Source.Execute
        Source.Executed -> PositionerSourceCopy.Execute
        PositionerSourceCopy.Executed -> PositionerSourceCopy2.Execute
        PositionerSourceCopy2.Executed -> Queue.Enqueue
        PlaneSensor.SensorOut -> Queue.Dequeue
        PlaneSensor.SensorOut -> SC_BeltConveyor.doPartInPos
        SimulationEvents.SimulationStarted -> Queue.Clear
        ParametricBoxLength_1.SizeY => Expression_with.boxwith
        Expression_with.Result => ParametricBoxLength_2.Transform.Y
        ParametricBoxLength_1.SizeX => ParametricBoxLength_2.SizeX
        ParametricBoxLength_1.SizeY => ParametricBoxLength_2.SizeY
        ParametricBoxLength_1.SizeZ => ParametricBoxLength_2.SizeZ
        ParametricBoxLength_1.SizeZ => Expression_height.boxheight
        Expression_height.Result => ParametricBoxLength_1.Transform.Z
        Expression_height.Result => ParametricBoxLength_2.Transform.Z
        ParametricBoxLength_1.SizeY => Expression_length.boxwith
        ParametricBoxLength_1.SizeY => Expression_with2.boxwith
        ParametricBoxLength_1.SizeY => ParametricBoxLeg.SizeY
        Expression_with.Result => MatrixRepeaterLegs.OffsetY
        ExpressionLegNumber.Result => SC_BeltConveyor.LegNumber
        SC_BeltConveyor.LegNumber => ExpressionLegOffset.LegNumber
        ExpressionLegOffset.Result => MatrixRepeaterLegs.OffsetX
        SC_BeltConveyor.LegNumber => ExpressionTotalLegNumber.LegNumber
        ExpressionTotalLegNumber.Result => MatrixRepeaterLegs.CountX
        Expression_with2.Result => ParametricCylinderRoller1.Height
        ParametricBoxLength_1.SizeY => ExpressionFootWith.BoxWith
        ParametricBoxLength_1.SizeY => ExpressionFootLength.BoxWith
        ExpressionFootWith.Result => ParametricBoxFoot.SizeX
        ExpressionFootLength.Result => ParametricBoxFoot.SizeY
        Expression_height.Result => ExpressionLegHeight.LegHeight
        ExpressionLegHeight.Result => ParametricBoxLeg.SizeZ
        ParametricBoxLength_1.SizeY => ExpressionFootYtransform.BoxWith
        ExpressionFootYtransform.Result => MatrixRepeaterFoots.Transform.Y
        ExpressionFootXtransform.Result => MatrixRepeaterFoots.Transform.X
        MatrixRepeaterLegs.CountX => MatrixRepeaterFoots.CountX
        MatrixRepeaterLegs.OffsetX => MatrixRepeaterFoots.OffsetX
        MatrixRepeaterLegs.OffsetY => ExpressionFootYoffset.LegOffsetY
        ParametricBoxLength_1.SizeY => ExpressionFootYoffset.BoxWith
        ExpressionFootYoffset.Result => MatrixRepeaterFoots.OffsetY
        ExpressionFootXtransform.Result => ParametricBoxFoot.Transform.X
        ExpressionFootYtransform.Result => ParametricBoxFoot.Transform.Y
        ParametricBoxLength_1.SizeY => ParametricCylinderRoller1.Transform.Y
        SC_BeltConveyor.FirstLegXpos => ExpressionLegNumber.FirstLegXtransform
        SC_BeltConveyor.FirstLegXpos => ExpressionLegOffset.FirstLegXtransform
        ParametricBoxLeg.SizeX => ExpressionLegXtransform.LegWith
        ParametricBoxLeg.SizeY => ExpressionLegCylinderYtransform.LegDepth
        ExpressionLegCylinderYtransform.Result => ParametricCylinderLeg.Transform.Y
        ParametricBoxFoot.SizeZ => ExpressionLegZtransform.FotHeght
        ExpressionLegZtransform.Result => MatrixRepeaterLegs.Transform.Z
        ExpressionLegZtransform.Result => ExpressionLegHeight.FootAndCylinder
        ExpressionLegZtransform.Result => ParametricBoxLeg.Transform.Z
        ExpressionTotalLegNumber.Result => MatrixRepeaterLegCylinders.CountX
        MatrixRepeaterLegs.OffsetX => MatrixRepeaterLegCylinders.OffsetX
        MatrixRepeaterLegs.OffsetY => MatrixRepeaterLegCylinders.OffsetY
        ExpressionLegCylinderYtransform.Result => MatrixRepeaterLegCylinders.Transform.Y
        ParametricBoxLeg.SizeY => ExpressionLegWith.LegDepth
        ExpressionLegWith.Result => ParametricBoxLeg.SizeX
        ParametricBoxFoot.SizeX => ExpressionFootXtransform.FootWith
        ParametricBoxFoot.SizeZ => MatrixRepeaterLegCylinders.Transform.Z
        ParametricBoxLength_1.SizeZ => ExpressionRollerRadius.BoxHeight
        ExpressionRollerRadius.Result => ExpressionRollerZoffset.RollerRadius
        ExpressionRollerZoffset.Result => ParametricCylinderRoller1.Transform.Z
        ExpressionRollerRadius.Result => ParametricCylinderRoller1.Radius
        ParametricBoxFoot.SizeZ => ParametricCylinderLeg.Transform.Z
        ExpressionLegZtransform.Result => ParametricCylinderLeg.Height
        ExpressionRollerRadius.Result => ExpressionRollerXtransform.RollerRadius
        ExpressionRollerXtransform.Result => ParametricCylinderRoller1.Transform.X
        ParametricCylinderRoller1.Height => ParametricCylinderRoller2.Height
        ParametricCylinderRoller1.Radius => ParametricCylinderRoller2.Radius
        ParametricBoxLength_1.SizeY => ParametricCylinderRoller2.Transform.Y
        ExpressionRollerZoffset.Result => ParametricCylinderRoller2.Transform.Z
        ExpressionRollerRadius.Result => ExpressionRooler2Xtransform.RollerRadius
        ExpressionRooler2Xtransform.Result => ParametricCylinderRoller2.Transform.X
        ExpressionRollerZoffset.Result => ExpressionBeltZtransform.RollerZtransform
        ExpressionRollerRadius.Result => ExpressionBeltZtransform.RollerRadius
        ExpressionBeltZtransform.Result => ParametricBoxBelt.Transform.Z
        ExpressionRollerRadius.Result => ExpressionRollerDiameter.RollerRadius
        ExpressionRollerDiameter.Result => ParametricBoxBelt.SizeZ
        ParametricCylinderRoller1.Height => ParametricBoxBelt.SizeY
        ExpressionRollerXtransform.Result => ParametricBoxBelt.Transform.X
        ParametricBoxLength_1.SizeY => ParametricBoxBelt.Transform.Y
        ExpressionRooler2Xtransform.Result => ExpressionBeltLength.Roller2Xtransform
        ExpressionRollerXtransform.Result => ExpressionBeltLength.Roller1Xtransform
        ExpressionBeltLength.Result => ParametricBoxBelt.SizeX
        SC_BeltConveyor.FirstLegXpos => MatrixRepeaterLegCylinders.Transform.X
        SC_BeltConveyor.FirstLegXpos => ParametricCylinderLeg.Transform.X
        SC_BeltConveyor.FirstLegXpos => ExpressionLegXtransform.CylLegPos
        SC_BeltConveyor.FirstLegXpos => ExpressionFootXtransform.FirstLegCylinderXtransform
        ExpressionLegXtransform.Result => MatrixRepeaterLegs.Transform.X
        ExpressionLegXtransform.Result => ParametricBoxLeg.Transform.X
        Source.Copy => PositionerSourceCopy.Object
        ParametricBoxLength_1.SizeY => VectorConverterCopyPos.Y
        ParametricBoxLength_1.SizeZ => VectorConverterCopyPos.Z
        VectorConverterCopyPos.Vector => PositionerSourceCopy2.Position
        PositionerSourceCopy.Object => PositionerSourceCopy2.Object
        PositionSensor.Position => PositionerSourceCopy.Position
        PositionSensor.Orientation => PositionerSourceCopy.Orientation
        Expression_length.Result => VectorConverterPlaneSensorOrigin.X
        ExpressionPlaneSensorHeight.Result => VectorConverterPlaneSensorOrigin.Z
        VectorConverterPlaneSensorOrigin.Vector => PlaneSensor.Origin
        VectorConverterPlaneSensorAxis2.Vector => PlaneSensor.Axis2
        Source.Copy => Queue.Back
        ExpressionCNVspeed.Result => LinearMover.Speed
        Queue.NumberOfObjects => ComparerObjectsInQueue.ValueA
        ExpressionLengthConverted.Result => ExpressionRooler2Xtransform.CNVlength
        ExpressionLengthConverted.Result => Expression_length.cnvlength
        ExpressionHeightConverted.Result => ExpressionPlaneSensorHeight.CNVheight
        ExpressionLengthConverted.Result => ExpressionLegNumber.CNVlength
        ExpressionWithConverted.Result => Expression_with2.cnvwith
        ExpressionHeightConverted.Result => Expression_height.cnvheight
        ExpressionWithConverted.Result => VectorConverterPlaneSensorAxis2.Y
        ExpressionHeightConverted.Result => ExpressionRollerZoffset.CNVheight
        ExpressionLengthConverted.Result => ExpressionLegOffset.CNVlength
        ExpressionWithConverted.Result => Expression_with.cnvwith
        ExpressionLengthConverted.Result => ParametricBoxLength_1.SizeX
        ParametricCylinderLeg.GeneratedPart => MatrixRepeaterUpdate.InValue10
        MatrixRepeaterUpdate.OutValue10 => MatrixRepeaterLegCylinders.Source
        ParametricCylinderRoller1.GeneratedPart => MatrixRepeaterUpdate.InValue13
        ParametricCylinderRoller2.GeneratedPart => MatrixRepeaterUpdate.InValue14
        ParametricBoxBelt.GeneratedPart => MatrixRepeaterUpdate.InValue15
        ParametricBoxFoot.GeneratedPart => MatrixRepeaterUpdate.InValue1
        MatrixRepeaterUpdate.OutValue1 => MatrixRepeaterFoots.Source
        ParametricBoxLength_1.GeneratedPart => MatrixRepeaterUpdate.InValue2
        ParametricBoxLeg.GeneratedPart => MatrixRepeaterUpdate.InValue3
        MatrixRepeaterUpdate.OutValue3 => MatrixRepeaterLegs.Source
        ParametricBoxLength_2.GeneratedPart => MatrixRepeaterUpdate.InValue4
        SC_BeltConveyor.Length => ExpressionLengthConverted.Length
        SC_BeltConveyor.Width => ExpressionWithConverted.With
        SC_BeltConveyor.Height => ExpressionHeightConverted.Height
        SC_BeltConveyor.SourceObject => Source.Source
        SC_BeltConveyor.ConveyorSpeed => ExpressionCNVspeed.ConveyorSpeed
    - ParametricBoxLength_1 [smart component, from Components\ParametricBox.rslib] at (0, 0, 370) mm
        properties: GeneratedPart=GeneratedPart; KeepGeometry=true; SizeX=3; SizeY=0.05; SizeZ=0.12
      - GeneratedPart [part], size 3000 x 50 x 120 mm
    - ParametricBoxLength_2 [smart component, from Components\ParametricBox.rslib] at (0, 350, 370) mm
        properties: GeneratedPart=GeneratedPart; KeepGeometry=true; SizeX=3; SizeY=0.05; SizeZ=0.12
      - GeneratedPart [part], size 3000 x 50 x 120 mm
    - Expression_with [smart component, from Components\Expression.rslib]
        properties: boxwith=0.05; cnvwith=0.4; Expression=cnvwith-boxwith; Result=0.35
    - Expression_height [smart component, from Components\Expression.rslib]
        properties: boxheight=0.12; cnvheight=0.5; Expression=cnvheight-boxheight-0,01; Result=0.37
    - Expression_length [smart component, from Components\Expression.rslib]
        properties: boxwith=0.05; cnvlength=3; Expression=cnvlength-boxwith; Result=2.95
    - Expression_with2 [smart component, from Components\Expression.rslib]
        properties: boxwith=0.05; cnvwith=0.4; Expression=cnvwith-(boxwith*2); Result=0.3
    - ParametricBoxLeg [smart component, from Components\ParametricBox.rslib] at (150, 0, 72) mm
        properties: GeneratedPart=GeneratedPart; KeepGeometry=true; SizeX=0.1; SizeY=0.05; SizeZ=0.298
      - GeneratedPart [part], size 100 x 50 x 298 mm
    - MatrixRepeaterLegs [smart component, from Components\MatrixRepeater.rslib] at (150, 0, 72) mm
        properties: CountX=2; CountY=2; CountZ=1; OffsetX=2.6; OffsetY=0.35; OffsetZ=0; Source=GeneratedPart
      - GeneratedPart [part], size 100 x 50 x 298 mm
      - GeneratedPart [part] at (2600, 0, 0) mm, size 100 x 50 x 298 mm
      - GeneratedPart [part] at (0, 350, 0) mm, size 100 x 50 x 298 mm
      - GeneratedPart [part] at (2600, 350, 0) mm, size 100 x 50 x 298 mm
    - ExpressionLegNumber [smart component, from Components\Expression.rslib]
        properties: CNVlength=3; Expression=(CNVlength-(FirstLegXtransform*2))/2,5; FirstLegXtransform=0.2; Result=1.04
    - ExpressionLegOffset [smart component, from Components\Expression.rslib]
        properties: CNVlength=3; Expression=(CNVlength-(FirstLegXtransform*2))/LegNumber; FirstLegXtransform=0.2; LegNumber=1; Result=2.6
    - ExpressionTotalLegNumber [smart component, from Components\Expression.rslib]
        properties: Expression=LegNumber+1; LegNumber=1; Result=2
    - ParametricCylinderRoller1 [smart component, from Components\ParametricCylinder.rslib] at (50, 50, 430) mm, rotated rx -90 ry 0 rz 0 deg
        properties: GeneratedPart=GeneratedPart; Height=0.3; KeepGeometry=true; Radius=0.07
      - GeneratedPart [part], size 140 x 138.6 x 300 mm
    - ParametricBoxFoot [smart component, from Components\ParametricBox.rslib] at (162.5, -50, 0) mm
        properties: GeneratedPart=GeneratedPart; KeepGeometry=true; SizeX=0.075; SizeY=0.1; SizeZ=0.012
      - GeneratedPart [part], size 75 x 100 x 12 mm
    - ExpressionFootWith [smart component, from Components\Expression.rslib]
        properties: BoxWith=0.05; Expression=BoxWith*1,5; Result=0.075
    - ExpressionFootLength [smart component, from Components\Expression.rslib]
        properties: BoxWith=0.05; Expression=BoxWith*2; Result=0.1
    - ExpressionLegHeight [smart component, from Components\Expression.rslib]
        properties: Expression=LegHeight-FootAndCylinder; FootAndCylinder=0.072; LegHeight=0.37; Result=0.298
    - MatrixRepeaterFoots [smart component, from Components\MatrixRepeater.rslib] at (162.5, -50, 0) mm
        properties: CountX=2; CountY=2; CountZ=1; OffsetX=2.6; OffsetY=0.4; OffsetZ=0.1; Source=GeneratedPart
      - GeneratedPart [part], size 75 x 100 x 12 mm
      - GeneratedPart [part] at (2600, 0, 0) mm, size 75 x 100 x 12 mm
      - GeneratedPart [part] at (0, 400, 0) mm, size 75 x 100 x 12 mm
      - GeneratedPart [part] at (2600, 400, 0) mm, size 75 x 100 x 12 mm
    - ExpressionFootYtransform [smart component, from Components\Expression.rslib]
        properties: BoxWith=0.05; Expression=-BoxWith; Result=-0.05
    - ExpressionFootXtransform [smart component, from Components\Expression.rslib]
        properties: Expression=FirstLegCylinderXtransform-(FootWith/2); FirstLegCylinderXtransform=0.2; FootWith=0.075; Result=0.1625
    - ExpressionFootYoffset [smart component, from Components\Expression.rslib]
        properties: BoxWith=0.05; Expression=LegOffsetY+BoxWith; LegOffsetY=0.35; Result=0.4
    - ParametricCylinderLeg [smart component, from Components\ParametricCylinder.rslib] at (200, 25, 12) mm
        properties: GeneratedPart=GeneratedPart; Height=0.072; KeepGeometry=true; Radius=0.01
      - GeneratedPart [part], size 20 x 19.7 x 72 mm
    - ExpressionLegXtransform [smart component, from Components\Expression.rslib]
        properties: CylLegPos=0.2; Expression=CylLegPos-(LegWith/2); LegWith=0.1; Result=0.15
    - ExpressionLegCylinderYtransform [smart component, from Components\Expression.rslib]
        properties: Expression=LegDepth/2; LegDepth=0.05; Result=0.025
    - ExpressionLegZtransform [smart component, from Components\Expression.rslib]
        properties: Expression=FotHeght+0,06; FotHeght=0.012; Result=0.072
    - MatrixRepeaterLegCylinders [smart component, from Components\MatrixRepeater.rslib] at (200, 25, 12) mm
        properties: CountX=2; CountY=2; CountZ=1; OffsetX=2.6; OffsetY=0.35; OffsetZ=0.1; Source=GeneratedPart
      - GeneratedPart [part], size 20 x 19.7 x 72 mm
      - GeneratedPart [part] at (2600, 0, 0) mm, size 20 x 19.7 x 72 mm
      - GeneratedPart [part] at (0, 350, 0) mm, size 20 x 19.7 x 72 mm
      - GeneratedPart [part] at (2600, 350, 0) mm, size 20 x 19.7 x 72 mm
    - ExpressionLegWith [smart component, from Components\Expression.rslib]
        properties: Expression=LegDepth*2; LegDepth=0.05; Result=0.1
    - ExpressionRollerRadius [smart component, from Components\Expression.rslib]
        properties: BoxHeight=0.12; Expression=(BoxHeight/2)+0,01; Result=0.07
    - ExpressionRollerZoffset [smart component, from Components\Expression.rslib]
        properties: CNVheight=0.5; Expression=CNVheight-RollerRadius; Result=0.43; RollerRadius=0.07
    - ExpressionRollerXtransform [smart component, from Components\Expression.rslib]
        properties: Expression=RollerRadius-0,02; Result=0.05; RollerRadius=0.07
    - ExpressionRooler2Xtransform [smart component, from Components\Expression.rslib]
        properties: CNVlength=3; Expression=CNVlength-(RollerRadius-0,02); Result=2.95; RollerRadius=0.0700000000000001
    - ParametricCylinderRoller2 [smart component, from Components\ParametricCylinder.rslib] at (2950, 50, 430) mm, rotated rx -90 ry 0 rz 0 deg
        properties: GeneratedPart=GeneratedPart; Height=0.3; KeepGeometry=true; Radius=0.07
      - GeneratedPart [part], size 140 x 138.6 x 300 mm
    - ParametricBoxBelt [smart component, from Components\ParametricBox.rslib] at (50, 50, 360) mm
        properties: GeneratedPart=GeneratedPart; KeepGeometry=true; SizeX=2.9; SizeY=0.3; SizeZ=0.14
      - GeneratedPart [part], size 2900 x 300 x 140 mm
    - ExpressionBeltZtransform [smart component, from Components\Expression.rslib]
        properties: Expression=RollerZtransform-RollerRadius; Result=0.36; RollerRadius=0.07; RollerZtransform=0.43
    - ExpressionRollerDiameter [smart component, from Components\Expression.rslib]
        properties: Expression=RollerRadius*2; Result=0.14; RollerRadius=0.07
    - ExpressionBeltLength [smart component, from Components\Expression.rslib]
        properties: Expression=Roller2Xtransform-Roller1Xtransform; Result=2.9; Roller1Xtransform=0.05; Roller2Xtransform=2.95
    - Source [smart component, from Components\Source.rslib]
        properties: Copy=(none); Orientation=[0 0 0]; Parent=(none); Position=[0 0 0]; Source=(none); Transient=false; PhysicsBehavior=-1
    - PositionerSourceCopy [smart component, from Components\Positioner.rslib]
        properties: Object=(none); Orientation=[0 0 0]; Position=[-1 0.1 0.37]; Reference=Global; ReferenceObject=(none)
    - PositionerSourceCopy2 [smart component, from Components\Positioner.rslib]
        properties: Object=(none); Orientation=[0 0 0]; Position=[0 0.05 0.12]; Reference=Local; ReferenceObject=(none)
    - VectorConverterCopyPos [smart component, from Components\VectorConverter.rslib]
        properties: Vector=[0 0.05 0.12]; X=0; Y=0.05; Z=0.12
    - PositionSensor [smart component, from Components\PositionSensor.rslib]
        properties: Object=ParametricBoxLength_1; Orientation=[0 0 0]; Position=[-1 0.1 0.37]; Reference=Global; ReferenceObject=(none)
    - PlaneSensor [smart component, from Components\PlaneSensor.rslib]
        properties: Axis1=[0 0 0.05]; Axis2=[0 0.4 0]; Origin=[2.95 0 0.51]; SensedPart=(none)
      - _sensorPart_ [part], size 0 x 400 x 50 mm
    - ExpressionPlaneSensorHeight [smart component, from Components\Expression.rslib]
        properties: CNVheight=0.5; Expression=CNVheight+0,01; Result=0.51
    - VectorConverterPlaneSensorOrigin [smart component, from Components\VectorConverter.rslib]
        properties: Vector=[2.95 0 0.51]; X=2.95; Y=0; Z=0.51
    - VectorConverterPlaneSensorAxis2 [smart component, from Components\VectorConverter.rslib]
        properties: Vector=[0 0.4 0]; X=0; Y=0.4; Z=0
    - Queue [smart component, from Components\Queue.rslib]
        properties: Back=(none); Front=(none); NumberOfObjects=0; Queue=
    - LinearMover [smart component, from Components\LinearMover.rslib]
        properties: Direction=[1 0 0]; Object=Queue; Reference=Local; ReferenceObject=(none); Speed=0.5
    - ExpressionCNVspeed [smart component, from Components\Expression.rslib]
        properties: ConveyorSpeed=500; Expression=ConveyorSpeed/1000; Result=0.5
    - SimulationEvents [smart component, from Components\SimulationEvents.rslib]
    - LogicGateSensorLow [smart component, from Components\LogicGate.rslib]
        properties: Delay=0; Operator=NOT
    - LogicGateNewPart [smart component, from Components\LogicGate.rslib]
        properties: Delay=0; Operator=AND
    - ComparerObjectsInQueue [smart component, from Components\Comparer.rslib]
        properties: Operator=<; ValueA=0; ValueB=1
    - LogicGateNewPart2 [smart component, from Components\LogicGate.rslib]
        properties: Delay=0; Operator=AND
    - ExpressionLengthConverted [smart component, from Components\Expression.rslib]
        properties: Expression=Length/1000; Length=3000; Result=3
    - ExpressionWithConverted [smart component, from Components\Expression.rslib]
        properties: Expression=With/1000; Result=0.4; With=400
    - ExpressionHeightConverted [smart component, from Components\Expression.rslib]
        properties: Expression=Height/1000; Height=500; Result=0.5
    - MatrixRepeaterUpdate [smart component, from %9EFD5320-513E-49BD-B6BC-92403559CEC9%\SC_BeltConveyor.rslib]
        properties: InValue1=GeneratedPart; InValue10=GeneratedPart; InValue11=(none); InValue12=(none); InValue13=GeneratedPart; InValue14=GeneratedPart; InValue15=GeneratedPart; InValue2=GeneratedPart; InValue3=GeneratedPart; InValue4=GeneratedPart; InValue5=(none); InValue6=(none); InValue7=(none); InValue8=(none); InValue9=(none); OutValue1=GeneratedPart; OutValue10=GeneratedPart; OutValue11=(none); OutValue12=(none); OutValue13=GeneratedPart; OutValue14=GeneratedPart; OutValue15=GeneratedPart; OutValue2=GeneratedPart; OutValue3=GeneratedPart; OutValue4=GeneratedPart; OutValue5=(none); OutValue6=(none); OutValue7=(none); OutValue8=(none); OutValue9=(none)
  - SC_BeltConveyor_1 [smart component, from %9EFD5320-513E-49BD-B6BC-92403559CEC9%\SC_BeltConveyor.rslib] at (-1000, -400, 0) mm
      properties: ConveyorSpeed=500; FirstLegXpos=0.2; Height=500; LegNumber=1; Length=3000; RollerNumber=31; SourceObject=(none); Width=400
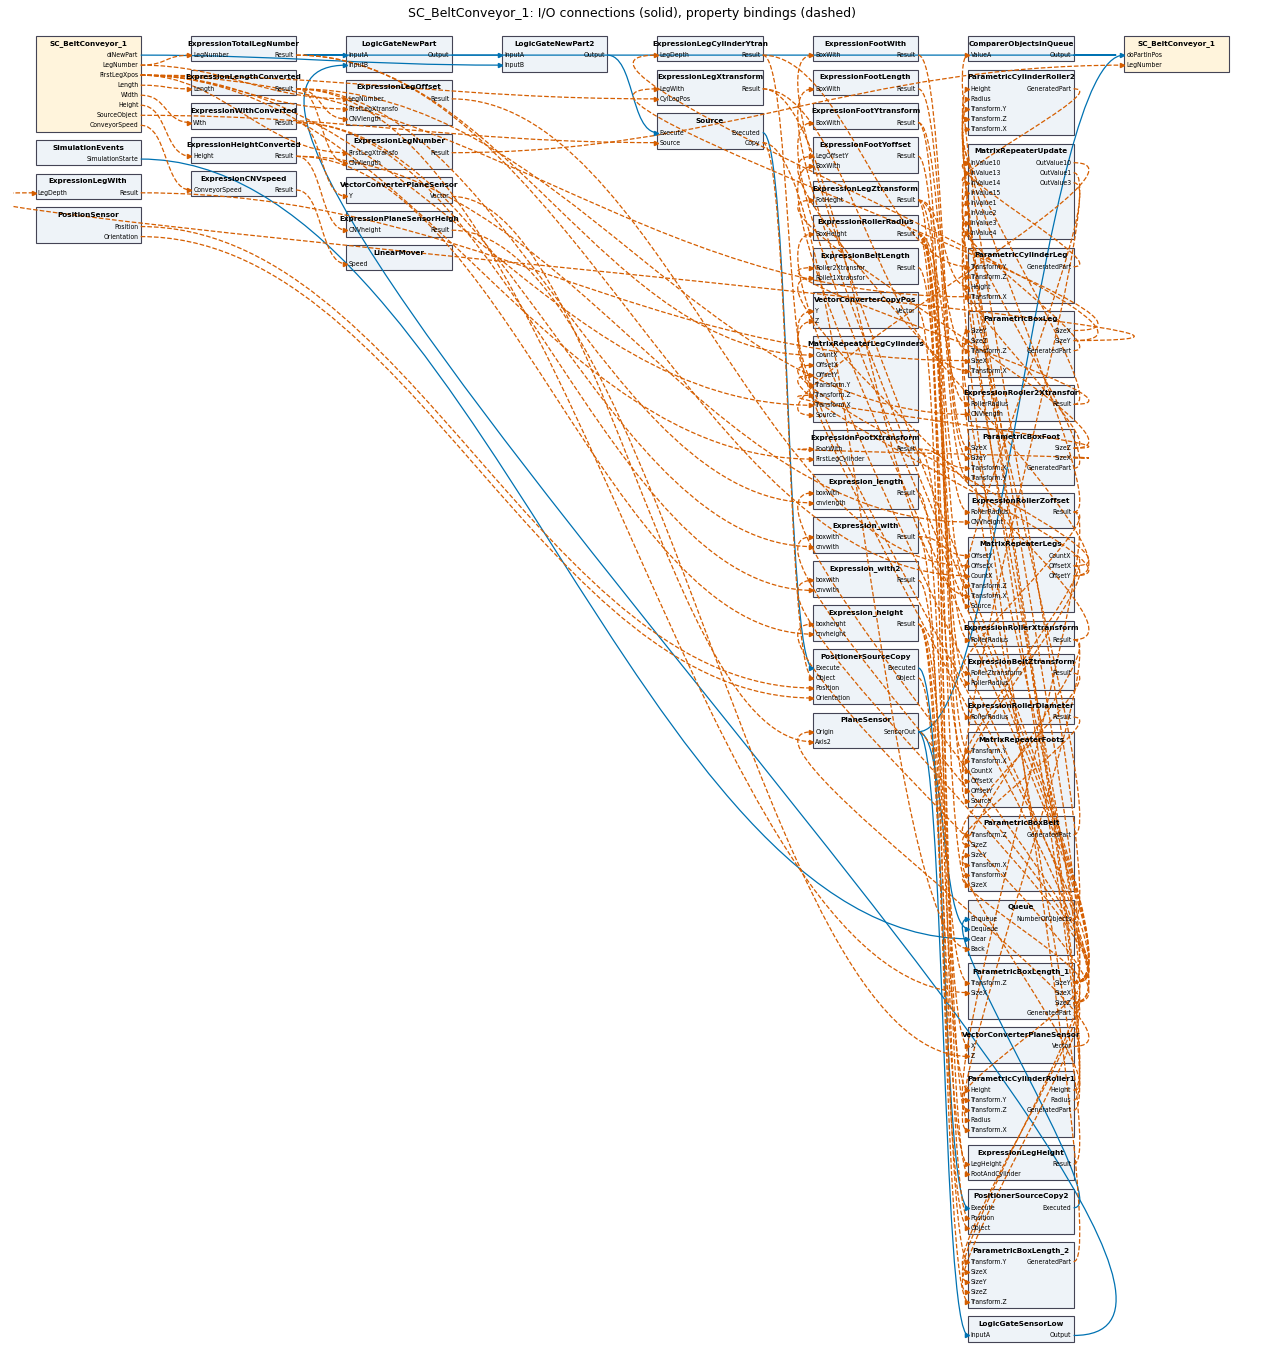
      connections:
        PlaneSensor.SensorOut -> LogicGateSensorLow.InputA
        ComparerObjectsInQueue.Output -> LogicGateNewPart.InputA
        LogicGateSensorLow.Output -> LogicGateNewPart.InputB
        LogicGateNewPart.Output -> LogicGateNewPart2.InputA
        SC_BeltConveyor_1.diNewPart -> LogicGateNewPart2.InputB
        LogicGateNewPart2.Output -> Source.Execute
        Source.Executed -> PositionerSourceCopy.Execute
        PositionerSourceCopy.Executed -> PositionerSourceCopy2.Execute
        PositionerSourceCopy2.Executed -> Queue.Enqueue
        PlaneSensor.SensorOut -> Queue.Dequeue
        PlaneSensor.SensorOut -> SC_BeltConveyor_1.doPartInPos
        SimulationEvents.SimulationStarted -> Queue.Clear
        ParametricBoxLength_1.SizeY => Expression_with.boxwith
        Expression_with.Result => ParametricBoxLength_2.Transform.Y
        ParametricBoxLength_1.SizeX => ParametricBoxLength_2.SizeX
        ParametricBoxLength_1.SizeY => ParametricBoxLength_2.SizeY
        ParametricBoxLength_1.SizeZ => ParametricBoxLength_2.SizeZ
        ParametricBoxLength_1.SizeZ => Expression_height.boxheight
        Expression_height.Result => ParametricBoxLength_1.Transform.Z
        Expression_height.Result => ParametricBoxLength_2.Transform.Z
        ParametricBoxLength_1.SizeY => Expression_length.boxwith
        ParametricBoxLength_1.SizeY => Expression_with2.boxwith
        ParametricBoxLength_1.SizeY => ParametricBoxLeg.SizeY
        Expression_with.Result => MatrixRepeaterLegs.OffsetY
        ExpressionLegNumber.Result => SC_BeltConveyor_1.LegNumber
        SC_BeltConveyor_1.LegNumber => ExpressionLegOffset.LegNumber
        ExpressionLegOffset.Result => MatrixRepeaterLegs.OffsetX
        SC_BeltConveyor_1.LegNumber => ExpressionTotalLegNumber.LegNumber
        ExpressionTotalLegNumber.Result => MatrixRepeaterLegs.CountX
        Expression_with2.Result => ParametricCylinderRoller1.Height
        ParametricBoxLength_1.SizeY => ExpressionFootWith.BoxWith
        ParametricBoxLength_1.SizeY => ExpressionFootLength.BoxWith
        ExpressionFootWith.Result => ParametricBoxFoot.SizeX
        ExpressionFootLength.Result => ParametricBoxFoot.SizeY
        Expression_height.Result => ExpressionLegHeight.LegHeight
        ExpressionLegHeight.Result => ParametricBoxLeg.SizeZ
        ParametricBoxLength_1.SizeY => ExpressionFootYtransform.BoxWith
        ExpressionFootYtransform.Result => MatrixRepeaterFoots.Transform.Y
        ExpressionFootXtransform.Result => MatrixRepeaterFoots.Transform.X
        MatrixRepeaterLegs.CountX => MatrixRepeaterFoots.CountX
        MatrixRepeaterLegs.OffsetX => MatrixRepeaterFoots.OffsetX
        MatrixRepeaterLegs.OffsetY => ExpressionFootYoffset.LegOffsetY
        ParametricBoxLength_1.SizeY => ExpressionFootYoffset.BoxWith
        ExpressionFootYoffset.Result => MatrixRepeaterFoots.OffsetY
        ExpressionFootXtransform.Result => ParametricBoxFoot.Transform.X
        ExpressionFootYtransform.Result => ParametricBoxFoot.Transform.Y
        ParametricBoxLength_1.SizeY => ParametricCylinderRoller1.Transform.Y
        SC_BeltConveyor_1.FirstLegXpos => ExpressionLegNumber.FirstLegXtransform
        SC_BeltConveyor_1.FirstLegXpos => ExpressionLegOffset.FirstLegXtransform
        ParametricBoxLeg.SizeX => ExpressionLegXtransform.LegWith
        ParametricBoxLeg.SizeY => ExpressionLegCylinderYtransform.LegDepth
        ExpressionLegCylinderYtransform.Result => ParametricCylinderLeg.Transform.Y
        ParametricBoxFoot.SizeZ => ExpressionLegZtransform.FotHeght
        ExpressionLegZtransform.Result => MatrixRepeaterLegs.Transform.Z
        ExpressionLegZtransform.Result => ExpressionLegHeight.FootAndCylinder
        ExpressionLegZtransform.Result => ParametricBoxLeg.Transform.Z
        ExpressionTotalLegNumber.Result => MatrixRepeaterLegCylinders.CountX
        MatrixRepeaterLegs.OffsetX => MatrixRepeaterLegCylinders.OffsetX
        MatrixRepeaterLegs.OffsetY => MatrixRepeaterLegCylinders.OffsetY
        ExpressionLegCylinderYtransform.Result => MatrixRepeaterLegCylinders.Transform.Y
        ParametricBoxLeg.SizeY => ExpressionLegWith.LegDepth
        ExpressionLegWith.Result => ParametricBoxLeg.SizeX
        ParametricBoxFoot.SizeX => ExpressionFootXtransform.FootWith
        ParametricBoxFoot.SizeZ => MatrixRepeaterLegCylinders.Transform.Z
        ParametricBoxLength_1.SizeZ => ExpressionRollerRadius.BoxHeight
        ExpressionRollerRadius.Result => ExpressionRollerZoffset.RollerRadius
        ExpressionRollerZoffset.Result => ParametricCylinderRoller1.Transform.Z
        ExpressionRollerRadius.Result => ParametricCylinderRoller1.Radius
        ParametricBoxFoot.SizeZ => ParametricCylinderLeg.Transform.Z
        ExpressionLegZtransform.Result => ParametricCylinderLeg.Height
        ExpressionRollerRadius.Result => ExpressionRollerXtransform.RollerRadius
        ExpressionRollerXtransform.Result => ParametricCylinderRoller1.Transform.X
        ParametricCylinderRoller1.Height => ParametricCylinderRoller2.Height
        ParametricCylinderRoller1.Radius => ParametricCylinderRoller2.Radius
        ParametricBoxLength_1.SizeY => ParametricCylinderRoller2.Transform.Y
        ExpressionRollerZoffset.Result => ParametricCylinderRoller2.Transform.Z
        ExpressionRollerRadius.Result => ExpressionRooler2Xtransform.RollerRadius
        ExpressionRooler2Xtransform.Result => ParametricCylinderRoller2.Transform.X
        ExpressionRollerZoffset.Result => ExpressionBeltZtransform.RollerZtransform
        ExpressionRollerRadius.Result => ExpressionBeltZtransform.RollerRadius
        ExpressionBeltZtransform.Result => ParametricBoxBelt.Transform.Z
        ExpressionRollerRadius.Result => ExpressionRollerDiameter.RollerRadius
        ExpressionRollerDiameter.Result => ParametricBoxBelt.SizeZ
        ParametricCylinderRoller1.Height => ParametricBoxBelt.SizeY
        ExpressionRollerXtransform.Result => ParametricBoxBelt.Transform.X
        ParametricBoxLength_1.SizeY => ParametricBoxBelt.Transform.Y
        ExpressionRooler2Xtransform.Result => ExpressionBeltLength.Roller2Xtransform
        ExpressionRollerXtransform.Result => ExpressionBeltLength.Roller1Xtransform
        ExpressionBeltLength.Result => ParametricBoxBelt.SizeX
        SC_BeltConveyor_1.FirstLegXpos => MatrixRepeaterLegCylinders.Transform.X
        SC_BeltConveyor_1.FirstLegXpos => ParametricCylinderLeg.Transform.X
        SC_BeltConveyor_1.FirstLegXpos => ExpressionLegXtransform.CylLegPos
        SC_BeltConveyor_1.FirstLegXpos => ExpressionFootXtransform.FirstLegCylinderXtransform
        ExpressionLegXtransform.Result => MatrixRepeaterLegs.Transform.X
        ExpressionLegXtransform.Result => ParametricBoxLeg.Transform.X
        Source.Copy => PositionerSourceCopy.Object
        ParametricBoxLength_1.SizeY => VectorConverterCopyPos.Y
        ParametricBoxLength_1.SizeZ => VectorConverterCopyPos.Z
        VectorConverterCopyPos.Vector => PositionerSourceCopy2.Position
        PositionerSourceCopy.Object => PositionerSourceCopy2.Object
        PositionSensor.Position => PositionerSourceCopy.Position
        PositionSensor.Orientation => PositionerSourceCopy.Orientation
        Expression_length.Result => VectorConverterPlaneSensorOrigin.X
        ExpressionPlaneSensorHeight.Result => VectorConverterPlaneSensorOrigin.Z
        VectorConverterPlaneSensorOrigin.Vector => PlaneSensor.Origin
        VectorConverterPlaneSensorAxis2.Vector => PlaneSensor.Axis2
        Source.Copy => Queue.Back
        ExpressionCNVspeed.Result => LinearMover.Speed
        Queue.NumberOfObjects => ComparerObjectsInQueue.ValueA
        ExpressionLengthConverted.Result => ExpressionRooler2Xtransform.CNVlength
        ExpressionLengthConverted.Result => Expression_length.cnvlength
        ExpressionHeightConverted.Result => ExpressionPlaneSensorHeight.CNVheight
        ExpressionLengthConverted.Result => ExpressionLegNumber.CNVlength
        ExpressionWithConverted.Result => Expression_with2.cnvwith
        ExpressionHeightConverted.Result => Expression_height.cnvheight
        ExpressionWithConverted.Result => VectorConverterPlaneSensorAxis2.Y
        ExpressionHeightConverted.Result => ExpressionRollerZoffset.CNVheight
        ExpressionLengthConverted.Result => ExpressionLegOffset.CNVlength
        ExpressionWithConverted.Result => Expression_with.cnvwith
        ExpressionLengthConverted.Result => ParametricBoxLength_1.SizeX
        ParametricCylinderLeg.GeneratedPart => MatrixRepeaterUpdate.InValue10
        MatrixRepeaterUpdate.OutValue10 => MatrixRepeaterLegCylinders.Source
        ParametricCylinderRoller1.GeneratedPart => MatrixRepeaterUpdate.InValue13
        ParametricCylinderRoller2.GeneratedPart => MatrixRepeaterUpdate.InValue14
        ParametricBoxBelt.GeneratedPart => MatrixRepeaterUpdate.InValue15
        ParametricBoxFoot.GeneratedPart => MatrixRepeaterUpdate.InValue1
        MatrixRepeaterUpdate.OutValue1 => MatrixRepeaterFoots.Source
        ParametricBoxLength_1.GeneratedPart => MatrixRepeaterUpdate.InValue2
        ParametricBoxLeg.GeneratedPart => MatrixRepeaterUpdate.InValue3
        MatrixRepeaterUpdate.OutValue3 => MatrixRepeaterLegs.Source
        ParametricBoxLength_2.GeneratedPart => MatrixRepeaterUpdate.InValue4
        SC_BeltConveyor_1.Length => ExpressionLengthConverted.Length
        SC_BeltConveyor_1.Width => ExpressionWithConverted.With
        SC_BeltConveyor_1.Height => ExpressionHeightConverted.Height
        SC_BeltConveyor_1.SourceObject => Source.Source
        SC_BeltConveyor_1.ConveyorSpeed => ExpressionCNVspeed.ConveyorSpeed
    - ParametricBoxLength_1 [smart component, from Components\ParametricBox.rslib] at (0, 0, 370) mm
        properties: GeneratedPart=GeneratedPart; KeepGeometry=true; SizeX=3; SizeY=0.05; SizeZ=0.12
      - GeneratedPart [part], size 3000 x 50 x 120 mm
    - ParametricBoxLength_2 [smart component, from Components\ParametricBox.rslib] at (0, 350, 370) mm
        properties: GeneratedPart=GeneratedPart; KeepGeometry=true; SizeX=3; SizeY=0.05; SizeZ=0.12
      - GeneratedPart [part], size 3000 x 50 x 120 mm
    - Expression_with [smart component, from Components\Expression.rslib]
        properties: boxwith=0.05; cnvwith=0.4; Expression=cnvwith-boxwith; Result=0.35
    - Expression_height [smart component, from Components\Expression.rslib]
        properties: boxheight=0.12; cnvheight=0.5; Expression=cnvheight-boxheight-0,01; Result=0.37
    - Expression_length [smart component, from Components\Expression.rslib]
        properties: boxwith=0.05; cnvlength=3; Expression=cnvlength-boxwith; Result=2.95
    - Expression_with2 [smart component, from Components\Expression.rslib]
        properties: boxwith=0.05; cnvwith=0.4; Expression=cnvwith-(boxwith*2); Result=0.3
    - ParametricBoxLeg [smart component, from Components\ParametricBox.rslib] at (150, 0, 72) mm
        properties: GeneratedPart=GeneratedPart; KeepGeometry=true; SizeX=0.1; SizeY=0.05; SizeZ=0.298
      - GeneratedPart [part], size 100 x 50 x 298 mm
    - MatrixRepeaterLegs [smart component, from Components\MatrixRepeater.rslib] at (150, 0, 72) mm
        properties: CountX=2; CountY=2; CountZ=1; OffsetX=2.6; OffsetY=0.35; OffsetZ=0; Source=GeneratedPart
      - GeneratedPart [part], size 100 x 50 x 298 mm
      - GeneratedPart [part] at (2600, 0, 0) mm, size 100 x 50 x 298 mm
      - GeneratedPart [part] at (0, 350, 0) mm, size 100 x 50 x 298 mm
      - GeneratedPart [part] at (2600, 350, 0) mm, size 100 x 50 x 298 mm
    - ExpressionLegNumber [smart component, from Components\Expression.rslib]
        properties: CNVlength=3; Expression=(CNVlength-(FirstLegXtransform*2))/2,5; FirstLegXtransform=0.2; Result=1.04
    - ExpressionLegOffset [smart component, from Components\Expression.rslib]
        properties: CNVlength=3; Expression=(CNVlength-(FirstLegXtransform*2))/LegNumber; FirstLegXtransform=0.2; LegNumber=1; Result=2.6
    - ExpressionTotalLegNumber [smart component, from Components\Expression.rslib]
        properties: Expression=LegNumber+1; LegNumber=1; Result=2
    - ParametricCylinderRoller1 [smart component, from Components\ParametricCylinder.rslib] at (50, 50, 430) mm, rotated rx -90 ry 0 rz 0 deg
        properties: GeneratedPart=GeneratedPart; Height=0.3; KeepGeometry=true; Radius=0.07
      - GeneratedPart [part], size 140 x 138.6 x 300 mm
    - ParametricBoxFoot [smart component, from Components\ParametricBox.rslib] at (162.5, -50, 0) mm
        properties: GeneratedPart=GeneratedPart; KeepGeometry=true; SizeX=0.075; SizeY=0.1; SizeZ=0.012
      - GeneratedPart [part], size 75 x 100 x 12 mm
    - ExpressionFootWith [smart component, from Components\Expression.rslib]
        properties: BoxWith=0.05; Expression=BoxWith*1,5; Result=0.075
    - ExpressionFootLength [smart component, from Components\Expression.rslib]
        properties: BoxWith=0.05; Expression=BoxWith*2; Result=0.1
    - ExpressionLegHeight [smart component, from Components\Expression.rslib]
        properties: Expression=LegHeight-FootAndCylinder; FootAndCylinder=0.072; LegHeight=0.37; Result=0.298
    - MatrixRepeaterFoots [smart component, from Components\MatrixRepeater.rslib] at (162.5, -50, 0) mm
        properties: CountX=2; CountY=2; CountZ=1; OffsetX=2.6; OffsetY=0.4; OffsetZ=0.1; Source=GeneratedPart
      - GeneratedPart [part], size 75 x 100 x 12 mm
      - GeneratedPart [part] at (2600, 0, 0) mm, size 75 x 100 x 12 mm
      - GeneratedPart [part] at (0, 400, 0) mm, size 75 x 100 x 12 mm
      - GeneratedPart [part] at (2600, 400, 0) mm, size 75 x 100 x 12 mm
    - ExpressionFootYtransform [smart component, from Components\Expression.rslib]
        properties: BoxWith=0.05; Expression=-BoxWith; Result=-0.05
    - ExpressionFootXtransform [smart component, from Components\Expression.rslib]
        properties: Expression=FirstLegCylinderXtransform-(FootWith/2); FirstLegCylinderXtransform=0.2; FootWith=0.075; Result=0.1625
    - ExpressionFootYoffset [smart component, from Components\Expression.rslib]
        properties: BoxWith=0.05; Expression=LegOffsetY+BoxWith; LegOffsetY=0.35; Result=0.4
    - ParametricCylinderLeg [smart component, from Components\ParametricCylinder.rslib] at (200, 25, 12) mm
        properties: GeneratedPart=GeneratedPart; Height=0.072; KeepGeometry=true; Radius=0.01
      - GeneratedPart [part], size 20 x 19.7 x 72 mm
    - ExpressionLegXtransform [smart component, from Components\Expression.rslib]
        properties: CylLegPos=0.2; Expression=CylLegPos-(LegWith/2); LegWith=0.1; Result=0.15
    - ExpressionLegCylinderYtransform [smart component, from Components\Expression.rslib]
        properties: Expression=LegDepth/2; LegDepth=0.05; Result=0.025
    - ExpressionLegZtransform [smart component, from Components\Expression.rslib]
        properties: Expression=FotHeght+0,06; FotHeght=0.012; Result=0.072
    - MatrixRepeaterLegCylinders [smart component, from Components\MatrixRepeater.rslib] at (200, 25, 12) mm
        properties: CountX=2; CountY=2; CountZ=1; OffsetX=2.6; OffsetY=0.35; OffsetZ=0.1; Source=GeneratedPart
      - GeneratedPart [part], size 20 x 19.7 x 72 mm
      - GeneratedPart [part] at (2600, 0, 0) mm, size 20 x 19.7 x 72 mm
      - GeneratedPart [part] at (0, 350, 0) mm, size 20 x 19.7 x 72 mm
      - GeneratedPart [part] at (2600, 350, 0) mm, size 20 x 19.7 x 72 mm
    - ExpressionLegWith [smart component, from Components\Expression.rslib]
        properties: Expression=LegDepth*2; LegDepth=0.05; Result=0.1
    - ExpressionRollerRadius [smart component, from Components\Expression.rslib]
        properties: BoxHeight=0.12; Expression=(BoxHeight/2)+0,01; Result=0.07
    - ExpressionRollerZoffset [smart component, from Components\Expression.rslib]
        properties: CNVheight=0.5; Expression=CNVheight-RollerRadius; Result=0.43; RollerRadius=0.07
    - ExpressionRollerXtransform [smart component, from Components\Expression.rslib]
        properties: Expression=RollerRadius-0,02; Result=0.05; RollerRadius=0.07
    - ExpressionRooler2Xtransform [smart component, from Components\Expression.rslib]
        properties: CNVlength=3; Expression=CNVlength-(RollerRadius-0,02); Result=2.95; RollerRadius=0.0700000000000001
    - ParametricCylinderRoller2 [smart component, from Components\ParametricCylinder.rslib] at (2950, 50, 430) mm, rotated rx -90 ry 0 rz 0 deg
        properties: GeneratedPart=GeneratedPart; Height=0.3; KeepGeometry=true; Radius=0.07
      - GeneratedPart [part], size 140 x 138.6 x 300 mm
    - ParametricBoxBelt [smart component, from Components\ParametricBox.rslib] at (50, 50, 360) mm
        properties: GeneratedPart=GeneratedPart; KeepGeometry=true; SizeX=2.9; SizeY=0.3; SizeZ=0.14
      - GeneratedPart [part], size 2900 x 300 x 140 mm
    - ExpressionBeltZtransform [smart component, from Components\Expression.rslib]
        properties: Expression=RollerZtransform-RollerRadius; Result=0.36; RollerRadius=0.07; RollerZtransform=0.43
    - ExpressionRollerDiameter [smart component, from Components\Expression.rslib]
        properties: Expression=RollerRadius*2; Result=0.14; RollerRadius=0.07
    - ExpressionBeltLength [smart component, from Components\Expression.rslib]
        properties: Expression=Roller2Xtransform-Roller1Xtransform; Result=2.9; Roller1Xtransform=0.05; Roller2Xtransform=2.95
    - Source [smart component, from Components\Source.rslib]
        properties: Copy=(none); Orientation=[0 0 0]; Parent=(none); Position=[0 0 0]; Source=(none); Transient=false; PhysicsBehavior=-1
    - PositionerSourceCopy [smart component, from Components\Positioner.rslib]
        properties: Object=(none); Orientation=[0 0 0]; Position=[-1 -0.4 0.37]; Reference=Global; ReferenceObject=(none)
    - PositionerSourceCopy2 [smart component, from Components\Positioner.rslib]
        properties: Object=(none); Orientation=[0 0 0]; Position=[0 0.05 0.12]; Reference=Local; ReferenceObject=(none)
    - VectorConverterCopyPos [smart component, from Components\VectorConverter.rslib]
        properties: Vector=[0 0.05 0.12]; X=0; Y=0.05; Z=0.12
    - PositionSensor [smart component, from Components\PositionSensor.rslib]
        properties: Object=ParametricBoxLength_1; Orientation=[0 0 0]; Position=[-1 -0.4 0.37]; Reference=Global; ReferenceObject=(none)
    - PlaneSensor [smart component, from Components\PlaneSensor.rslib]
        properties: Axis1=[0 0 0.05]; Axis2=[0 0.4 0]; Origin=[2.95 0 0.51]; SensedPart=(none)
      - _sensorPart_ [part], size 0 x 400 x 50 mm
    - ExpressionPlaneSensorHeight [smart component, from Components\Expression.rslib]
        properties: CNVheight=0.5; Expression=CNVheight+0,01; Result=0.51
    - VectorConverterPlaneSensorOrigin [smart component, from Components\VectorConverter.rslib]
        properties: Vector=[2.95 0 0.51]; X=2.95; Y=0; Z=0.51
    - VectorConverterPlaneSensorAxis2 [smart component, from Components\VectorConverter.rslib]
        properties: Vector=[0 0.4 0]; X=0; Y=0.4; Z=0
    - Queue [smart component, from Components\Queue.rslib]
        properties: Back=(none); Front=(none); NumberOfObjects=0; Queue=
    - LinearMover [smart component, from Components\LinearMover.rslib]
        properties: Direction=[1 0 0]; Object=Queue; Reference=Local; ReferenceObject=(none); Speed=0.5
    - ExpressionCNVspeed [smart component, from Components\Expression.rslib]
        properties: ConveyorSpeed=500; Expression=ConveyorSpeed/1000; Result=0.5
    - SimulationEvents [smart component, from Components\SimulationEvents.rslib]
    - LogicGateSensorLow [smart component, from Components\LogicGate.rslib]
        properties: Delay=0; Operator=NOT
    - LogicGateNewPart [smart component, from Components\LogicGate.rslib]
        properties: Delay=0; Operator=AND
    - ComparerObjectsInQueue [smart component, from Components\Comparer.rslib]
        properties: Operator=<; ValueA=0; ValueB=1
    - LogicGateNewPart2 [smart component, from Components\LogicGate.rslib]
        properties: Delay=0; Operator=AND
    - ExpressionLengthConverted [smart component, from Components\Expression.rslib]
        properties: Expression=Length/1000; Length=3000; Result=3
    - ExpressionWithConverted [smart component, from Components\Expression.rslib]
        properties: Expression=With/1000; Result=0.4; With=400
    - ExpressionHeightConverted [smart component, from Components\Expression.rslib]
        properties: Expression=Height/1000; Height=500; Result=0.5
    - MatrixRepeaterUpdate [smart component, from %9EFD5320-513E-49BD-B6BC-92403559CEC9%\SC_BeltConveyor.rslib]
        properties: InValue1=GeneratedPart; InValue10=GeneratedPart; InValue11=(none); InValue12=(none); InValue13=GeneratedPart; InValue14=GeneratedPart; InValue15=GeneratedPart; InValue2=GeneratedPart; InValue3=GeneratedPart; InValue4=GeneratedPart; InValue5=(none); InValue6=(none); InValue7=(none); InValue8=(none); InValue9=(none); OutValue1=GeneratedPart; OutValue10=GeneratedPart; OutValue11=(none); OutValue12=(none); OutValue13=GeneratedPart; OutValue14=GeneratedPart; OutValue15=GeneratedPart; OutValue2=GeneratedPart; OutValue3=GeneratedPart; OutValue4=GeneratedPart; OutValue5=(none); OutValue6=(none); OutValue7=(none); OutValue8=(none); OutValue9=(none)
  - Basler Scout [part, from %048999B1-D959-4DC3-83C2-40272953C96E%\Basler Scout.rslib] at (-600, 300, 1000) mm
  - PlaneSensor [smart component, from %EB5A83E1-0387-4153-A644-55003E611B0E%\PlaneSensor.rslib] at (-600, -390, 502) mm, rotated rx 0 ry 0 rz 90 deg
      properties: Origin=[0 0 0]; Axis1=[0.38 0 0]; Axis2=[0 0 0.1]; SensedPart=MainBody
    - _sensorPart_ [part], size 380 x 0 x 100 mm
  - IRB360_1_1600_4D_STD_3 [mechanism, from Robots\IRB360_1_1600_4D_STD_02.rslib] at (1200, 0, 1800) mm, rotated rx 180 ry 0 rz 0 deg; joint values [0, 0, 0, 0] (rad or m)
  - ConveyorMechanism_2 [mechanism, from %3FC1A3B3-DC1B-42D2-8AA6-D9E1B3C46536%\PMConveyorMechanism.rslib] at (0, 0, 0) mm
  - ConveyorMechanism_3 [mechanism, from %3FC1A3B3-DC1B-42D2-8AA6-D9E1B3C46536%\PMConveyorMechanism.rslib] at (0, 0, 0) mm
  - Vacuum 1x1_1 [part, from %C4396042-08E9-4F2C-9889-A5FB4C9DA8F9%\Vacuum 1x1.rslib] at (1200, 0, 545.63) mm, rotated rx 180 ry 0 rz 0 deg
Attachment: Vacuum 1x1 is attached to IRB360_1_1600_4D_STD_02 / RevoluteLinkPlate
Attachment: Basler Scout is attached to SC_BeltConveyor
Attachment: PlaneSensor is attached to SC_BeltConveyor_1
Attachment: Vacuum 1x1_1 is attached to IRB360_1_1600_4D_STD_3 / RevoluteLinkPlate
Attachment: PickPlaceTool_1 is attached to IRB360_1_1600_4D_STD_02 / RevoluteLinkPlate
Attachment: PickPlaceTool_2 is attached to IRB360_1_1600_4D_STD_3 / RevoluteLinkPlate
Attachment: Vision_1 is attached to Basler Scout
Attachment: Camera 1 is attached to Basler Scout
Station logic (signal -> signal, property => property):
  Controller4.cnv1_doTrigVis -> Vision_1.TrigVisionIn
  Controller4.cnv1_doStartCnv -> Conveyor_1.CnvStartStopIn
  Controller4.CNV1_goCntSim -> ConveyorWorkArea_1.Cnt1ToEncIn
  Controller4.c1CntToEncStr -> ConveyorWorkArea_1.CntToEncStrobeIn
  Controller4.c1WaitWObj -> ConveyorWorkArea_1.WaitWobjIn
  Controller4.c1DropWObj -> ConveyorWorkArea_1.DropWobjIn
  Controller4.cnv1_doQIdle -> ConveyorWorkArea_1.QueueIdleIn
  Controller4.cnv2_doTrigVis -> Predefined_1.PosGenIn
  Controller4.cnv2_doStartCnv -> Conveyor_2.CnvStartStopIn
  Controller4.CNV2_goCntSim -> ConveyorWorkArea_1.Cnt1ToEncIn
  Controller4.c2CntToEncStr -> ConveyorWorkArea_1.CntToEncStrobeIn
  Controller4.c2WaitWObj -> ConveyorWorkArea_1.WaitWobjIn
  Controller4.c2DropWObj -> ConveyorWorkArea_1.DropWobjIn
  Controller4.cnv2_doQIdle -> ConveyorWorkArea_1.QueueIdleIn
  Controller4.doVacuum1 -> PickPlaceTool_1.GripIn
  Controller4.doBlow1 -> PickPlaceTool_1.ReleaseIn
  PlaneSensor.SensorOut -> Predefined_1.PosGenIn
